//
// Next Step
//
//   Switch over to next step under conditions:
//   or Maximal steptime
//   or Minimal steptime
//           and
//               or no setpoint delta temp
//               or atual value delta temp is ge setpoint deltatemp
//                   and sensor is ok
//           and
// /              or no setpoint max temp above floor
//              or atual value max temp above floor is ge setpoint max temp above floor
//                  and sensor is ok
// 1 Kriterium
      U(    ;
      L     "MAL1S033Par".ActTimeStepProcess.SteptimeActMinOverall; // Steptime in min overall
      L     "MAL1S033Par".StepAct.StepTime_Max; // Target steptime actual step
      >=I   ;
      )     ;
      O(    ;
// 2 Kriterium
      O(    ;
      U(    ;
      L     "MAL1S033Par".StepAct.DeltaTempSwitchpointStep;
      L     0;
//JV230310      >=D
      >D    ; //JV230310
      )     ;
// condition, if analogue input is not damaaged   //
      UN    "G295M".A_3291_BTE07.OutOverflow; //AIR TEMPERATURE ABOVE FLOOR
      UN    "G295M".A_3291_BTE07.OutFaultAI; //AIR TEMPERATURE ABOVE FLOOR
      UN    "G295M".A_3291_BTE01.OutOverflow; //AIR TEMPERATURE BELOW FLOOR
      UN    "G295M".A_3291_BTE01.OutFaultAI; //AIR TEMPERATURE BELOW FLOOR
      U(    ;
      L     "G295M".A_3291_BTE01.OutValueUnits; // act value temperature below floor
      L     "G295M".A_3291_BTE07.OutValueUnits; // act value temperature above floor
      -D    ; // delta temp actual
      L     L#10;
      /D    ;
      L     "MAL1S033Par".StepAct.DeltaTempSwitchpointStep;
      <D    ;
      )     ;
      )     ;
// 3 Kriterium
      O(    ;
      U(    ;
      L     "MAL1S033Par".StepAct.MaxTempAboveFloorStep;
      L     L#0; // 0,0°C is illegally switchpoint for max. temperature
      >D    ;
      )     ;
// condition, if analogue input is not damaaged   // MW R2.1
      UN    "G295M".A_3291_BTE01.OutOverflow; //AIR TEMPERATURE BELOW FLOOR
      UN    "G295M".A_3291_BTE01.OutFaultAI; //AIR TEMPERATURE BELOW FLOOR
      U(    ;
      L     "G295M".A_3291_BTE07.OutValueUnits; // act value temperature above floor
      L     L#10;
      /D    ;
      L     "MAL1S033Par".StepAct.MaxTempAboveFloorStep;
      >=D   ;
      )     ;
      )     ;
// 4 Kriterium
// and min. time
      U(    ;
      L     "MAL1S033Par".ActTimeStepProcess.SteptimeActMinOverall; // Steptime in min overall
//JV210710 Unsinn      L     "MAL1S033Par".RecipeHeader.Cleaning.SPARE_INT0001    // Target steptime actual step
      L     "MAL1S033Par".StepAct.StepTime_Min; // Target steptime actual step //JV210710
      >=I   ;
      )     ;
      )     ;
// and not cooling                                // UK 22.01.07
      UN    "MAL1S033Par".Par.FlagProcess.Cooling_Activ;
// 5 Kriterium
      O(    ;
      U     "MAL1S033Par".Par.FlagProcess.Cooling_Activ;
      U(    ;
      L     "G295M".A_3291_BTE07.OutValueUnits; // act value temperature above floor
      L     L#10;
      /D    ;
      L     "MAL1S033Par".StepAct.TemperaturAboveFloor;
      <=D   ;
      )     ;
      O(    ;
      L     "MAL1S033Par".Par.ParIntMachine.ActualStep;
//JV210710      L     25                          // max. 24 Schritte
      L     27; // max. 26 Schritte   //JV210710
      >=I   ;
      )     ;
      )     ;
// and min. time
      U(    ;
      L     "MAL1S033Par".ActTimeStepProcess.SteptimeActMinOverall; // Steptime in min overall
      L     "MAL1S033Par".StepAct.StepTime_Min; // Target steptime actual step
      >=I   ;
      )     ;
      SPBN  E606;
// send average step data to PIC
      SET   ;
      S     "MAL1S033StepValues".SendData; // send average step data to PIC
// Next step
      L     "MAL1S033Par".Par.ParIntMachine.ActualStep;
      L     "MAL1S033Par".RecipeHeader.NumberOfSteps;
      >I    ;
      SPB   Pedk; // Last step is finished
//BRT20100901 ====> Schritt halten
      U     "MAL1S033Par".Par.FlagProcess.Inf08; // Schritt halten
      SPB   E606;
//BRT20100901 <====
//
      L     "MAL1S033Par".Par.ParIntMachine.ActualStep;
      L     1;
      +I    ;
      T     "MAL1S033Par".Par.ParIntMachine.ActualStep;
      L     0;
      T     "MAL1S033Par".ActTimeStepProcess.SteptimeActMinOverall; // Steptime in min Overall
      SPA   E606;
Pedk: NOP   0; // Process has finished
      SET   ;
      R     "MAL1S033Par".Par.FlagProcess.ProcessActive;
      R     "MAL1S033Par".Par.FlagProcess.Cooling_Activ;
      S     "MAL1S033Par".Par.FlagProcess.ProcessEnd;
//
      L     0; // clear step number
      T     "MAL1S033Par".Par.ParIntMachine.ActualStep;
      T     "MAL1S033Par".StepAct.StepNumber;
E606: NOP   0;
NETWORK
TITLE =ASW_6080: Active step kilning
//
      U     "MAL1S033Par".Par.FlagProcess.ProcessActive;
      SPBN  E608;
// copy stepnr for visu
      L     "MAL1S033Par".Par.ParIntMachine.ActualStep;
      T     "MAL1S033Par".Par.ParIntProcess.ActualStep;
//MW 2010.04.26
      U(    ;
      L     "MAL1S033Par".StepAct.StepTime_Min;
      L     0;
      ==I   ;
      )     ;
      U(    ;
      L     "MAL1S033Par".StepAct.StepTime_Max;
      L     0;
      ==I   ;
      )     ;
      SPB   Nklk;
// basic speed  fans
      L     "MAL1S033Par".StepAct.SpeedVentilatorBasic;
      T     "MAL1S033Par".Par.ParIntProcess.SpeedVentilatorBasic;
// basic position exhaust air flaps
      L     "MAL1S033Par".StepAct.PosExhaustAirFlapBasic; // setpoint from recipe
      L     10; // convert to 0.1%
      *I    ;
      T     "MAL1S033Par".Par.ParIntProcess.PosExhaustAirFlapBasic;
// basic position withering air channel flaps
      L     "MAL1S033Par".StepAct.PosWitheringAirFlapBasic; // setpoint from recipe
      L     10; // convert to 0.1%
      *I    ;
      T     "MAL1S033Par".Par.ParIntProcess.PosWitheringAirFlapBasic;
// basic position recycling air channel flaps
      L     "MAL1S033Par".StepAct.PosRecycleAirFlapBasic; // setpoint from recipe
      L     10; // convert to 0.1%
      *I    ;
      T     "MAL1S033Par".Par.ParIntProcess.PosRecycAirFlapBasic;
      T     "MAL1S033Par".Par.ProcessValue.Value17; // Sollwert Umluftklappen Verbund
//MW 2010.04.26
// basic position fresh air flaps
//      L     "MAL1S033Par".StepAct.PosFreshAirFlapBasic    // setpoint from recipe
      L     0; // 0%
      U     "MAL1S033Par".Par.FlagProcess.ProcessActive;
      UN    "MAL1S033Par".Par.FlagProcess.Cooling_Activ;
      SPB   klk;
      L     100; // 100%
      U     "MAL1S033Par".Par.FlagProcess.ProcessActive;
      U     "MAL1S033Par".Par.FlagProcess.Cooling_Activ;
      SPB   klk;
      SPA   Nklk;
klk:  L     10; // convert to 0.1%
      *I    ;
      T     "MAL1S033Par".Par.ParIntProcess.PosFreshAirFlapBasic;
Nklk: NOP   0;

// Nachlauf der Brenner
//    U     "GCS7_GrCtrlDB".OutEnable[276]    // G276M Heating Kilningbox
      U     "MAL1S033Par".Par.FlagProcess.ProcessActive;
      UN    "MAL1S033Par".Par.FlagProcess.Cooling_Activ;
      =     "MAL1S033Par".Par.FlagProcess.ProgrammSchwelkenDarren;

      U     "MAL1S033Par".Par.FlagProcess.ProgrammSchwelkenDarren;
      L     S5T#1M;
      SA    T     60; // Nachlauf Brenner

      UN    "MAL1S033Par".Par.FlagProcess.ProgrammSchwelkenDarren;
      U     T     60; // Nachlauf Brenner
      =     "MAL1S033Par".Par.FlagProcess1.HilfsRegler_1_Down;
      =     "MAL1S033Par".Par.FlagProcess1.HilfsRegler_2_Down;
      =     "MAL1S033Par".Par.FlagProcess1.HilfsRegler_3_Down;
      =     "MAL1S033Par".Par.FlagProcess1.HilfsRegler_4_Down;

// Sollwert - Istwert vergleich der Temperatur unter der Horde
      L     "MAL1S033Par".StepAct.TemperaturBelowFloor; // setpoint from SCADA
      L     L#10;
      *D    ;
      T     "MAL1S033Par".Par.ProcessValue.TemperaturBelowFloor;

      U     "SYS_Scan0_Tick1min";
      SPBN  NORM;
//- nur alle x Minuten korrigieren ---
      L     "MAL1S033Par".Par.ProcessValue.CorrInterval;
      +     1;
      T     "MAL1S033Par".Par.ProcessValue.CorrInterval;
      L     2; // Korrekturintervall [min]
      >=I   ;
      SPBN  NORM;
      L     0;
      T     "MAL1S033Par".Par.ProcessValue.CorrInterval;

      L     "MAL1S033Par".Par.ProcessValue.TemperaturBelowFloor;
      L     "G295M".A_3291_BTE01.OutValueUnits; // Real-Value Temperature below floor
      -D    ;
      L     50; // Totband in [0.5°C]
      <=D   ;
      SPB   uebe; // wenn größer keine Korrektur
//- zur Sicherheit nicht mehr als 5.0°C zulassen ---
      L     5.000000e+002; // max. Korrektur !
      L     "MAL1S033Par".Par.ProcessValue_Real.SollwertTempKorr;
      <=R   ;
      SPB   uebe;
      L     "MAL1S033Par".Par.ProcessValue_Real.SollwertTempKorr;
      L     1.000000e+000; // Anpassung an Differenz zwischen den PT100
      +R    ;
      T     "MAL1S033Par".Par.ProcessValue_Real.SollwertTempKorr;
uebe: NOP   0;

      L     "MAL1S033Par".Par.ProcessValue.TemperaturBelowFloor;
      L     "G295M".A_3291_BTE01.OutValueUnits; // Real-Value Temperature below floor
      -D    ;
      L     50; // Totband in [0.5°C]
      >=D   ;
      SPB   unte; // wenn kleier keine Korrektur
//- keine negative Korrektur (führt sonst zu Schwingung) ---
      L     0.000000e+000; // keine negative Korrektur !
      L     "MAL1S033Par".Par.ProcessValue_Real.SollwertTempKorr;
      >=R   ;
      SPB   unte;
      L     1.000000e+000; // Anpassung an Differenz zwischen den PT100
      -R    ;
      T     "MAL1S033Par".Par.ProcessValue_Real.SollwertTempKorr;
unte: NOP   0;

//- bei Schrittbegin noch keine Korrektur ---
NORM: L     "MAL1S033Par".ActTimeStepProcess.SteptimeActMinOverall; // Steptime in min overall
      L     8; // Korrekturverzögerung [min]
      >I    ;
      SPB   SET;
      L     0.000000e+000;
      T     "MAL1S033Par".Par.ProcessValue_Real.SollwertTempKorr;
      L     10; // grossen Wert in Intervallzähler vorladen ...
      T     "MAL1S033Par".Par.ProcessValue.CorrInterval; // ... damit nächster 1MinTick gleich wirksam wird

SET:  NOP   0;
      L     "MAL1S033Par".Par.ProcessValue.TemperaturBelowFloor;
      DTR   ;
      L     "MAL1S033Par".Par.ProcessValue_Real.SollwertTempKorr;
      +R    ;
      T     "MAL1S033Par".Par.ProcessValue_Real.T_SOLL_NORM;
      SPA   M641;
      NOP   0;
//- Korrekturfaktor auf "0" setzen ---
      L     0.000000e+000;
      T     "MAL1S033Par".Par.ProcessValue_Real.SollwertTempKorr;
M641: NOP   0;
      SPA   GCPR;

// GCPRO
// setpoint temperature below floor
      NOP   0; // setpoint fans automatic mode
      L     L#0;
      U     "MAL1S033Par".Par.FlagProcess.Cooling_Activ; // switch over to cooling
      SPB   aut1;
      L     "MAL1S033Par".StepAct.TemperaturBelowFloor; // setpoint from SCADA
aut1: NOP   0;
      DTR   ;
      L     1.000000e+001;
      /R    ;
      T     "MAL1S033Par".Par.ProcessValue_Real.T_SOLL_NORM;
// emergency kiln heating
// fan 1
      U(    ;
      L     2#1;
      L     "MAL1S033Par".RecipeHeader.DeselectVentilator; // emergency regime without fan 1
      ==I   ;
      )     ;
      L     "G295M".A_3291_BTE05.OutValuePc; //AIR TEMPERATURE DIFFUSOR FAN 1 :  temperature in diffusor fan 1
      SPBN  c1R1;
      L     "G295M".A_3291_BTE01.OutValuePc; //AIR TEMPERATURE BELOW FLOOR
      L     "G295M".A_3291_BTE05.OutValuePc; //AIR TEMPERATURE DIFFUSOR FAN 1 :  temperature in diffusor fan 2
      <D    ;
      SPBN  c1R1;
      TAK   ;
c1R1: T     "MAL1S033Par".Par.ParIntProcess.ActValueTemperature_R1;
// fan 2
      U(    ;
      L     2#10;
      L     "MAL1S033Par".RecipeHeader.DeselectVentilator; // emergency regime without fan 2
      ==I   ;
      )     ;
      L     "G295M".A_3291_BTE05.OutValuePc; //AIR TEMPERATURE DIFFUSOR FAN 1 :  temperature in diffusor fan 2
      SPBN  c1R2;
      L     "G295M".A_3291_BTE01.OutValuePc; //AIR TEMPERATURE BELOW FLOOR
      L     "G295M".A_3291_BTE05.OutValuePc; //AIR TEMPERATURE DIFFUSOR FAN 1 :  temperature in diffusor fan 1
      <D    ;
      SPBN  c1R2;
      TAK   ;
c1R2: T     "MAL1S033Par".Par.ParIntProcess.ActValueTemperature_R2;

GCPR: NOP   0;
//BRT20100901 ====> Schritt halten, wenn in Rezept aktiviert!!!
      U(    ;
      L     "MAL1S033Par".RecipeHeader.SPARE_DINT004;
      L     L#1; // Schritt halten aktiviert = 1
      ==D   ;
      )     ;
      U(    ;
      L     "G295M".A_3291_BTE07.OutValuePc; // Temperature above floor kiln 2
      L     100;
      /D    ;
      L     "MAL1S033Par".RecipeHeader.SPARE_INT002; // Schaltpunkt für Schritt halten
      >=I   ;
      )     ;
      U(    ;
      U     "MAL1S032".ToASW.InfDataReady; // Kiln 1 bereit
      O     "MAL1S032Par".Par.FlagFunction_1.StepLoading;
      )     ;
      UN    "MAL1S032Par".Par.FlagProcess.ProcessActive;
      UN(   ;
      U     "G271M".A_3125_MXZ01MA.Ma.StStartedFwd;
      U     "G271M".A_3125_TSC01_AF.OutL; // Ventilator 1 dreht mind. 40% SW
      U     "G271M".A_3126_MXZ01MA.Ma.StStartedFwd;
      U     "G271M".A_3126_TSC01_AF.OutL; // Ventilator 2 dreht mind. 40% SW
      )     ;
      S     "MAL1S033Par".Par.FlagProcess.Inf08; // Schritt halten

      U(    ;
      L     "MAL1S033Par".RecipeHeader.SPARE_DINT004;
      L     L#1; // Schritt halten aktiviert = 1
      <>D   ;
      )     ;
      O(    ;
      U     "MAL1S032Par".Par.FlagProcess.ProcessActive;
      U(    ;
      U     "G271M".A_3125_MXZ01MA.Ma.StStartedFwd;
      U     "G271M".A_3125_TSC01_AF.OutL; // Ventilator 1 dreht mind. 40% SW
      O     ;
      U     "G271M".A_3126_MXZ01MA.Ma.StStartedFwd;
      U     "G271M".A_3126_TSC01_AF.OutL; // Ventilator 2 dreht mind. 40% SW
      )     ;
      )     ;
      R     "MAL1S033Par".Par.FlagProcess.Inf08; // Schritt halten
//BRT20100901 <====
// cooling down
      L     "MAL1S033Par".StepAct.CoolingDown;
      L     1;
      ==I   ;
      S     "MAL1S033Par".Par.FlagProcess.Cooling_Activ;
//JV250710 =====>
      L     "MAL1S033Par".Par.ParIntMachine.ActualStep;
      L     24;
      <I    ;
      O(    ; //JV290710 ======>
      L     "MAL1S033Par".StepAct.CoolingDown;
      L     1;
      <>I   ;
      )     ; //JV290710 <=====
      R     "MAL1S033Par".Par.FlagProcess.Cooling_Activ;
//JV250710 <=====
E608: NOP   0;
//BRT20100901 ====> Schritt-Halte-Bit wird nochmals explizit bei Prozess Ende zurückgesetzt!!!
      UN    "MAL1S033Par".Par.FlagProcess.ProcessActive;
      O     "MAL1S033Par".Par.FlagProcess.ProcessEnd;
      R     "MAL1S033Par".Par.FlagProcess.Inf08; // Schritt halten

// Abdarr-Betrieb aktiv
      U(    ;
      L     "MAL1S033Par".Par.ParIntMachine.ActualStep;
      L     "MAL1S032Par".Par.ParIntMachine.ActualStep;
      >I    ;
      )     ;
      UN    "MAL1S033Par".Par.FlagProcess.Cooling_Activ;
      O     "MAL1S032Par".Par.FlagProcess.Cooling_Activ;
//BRT20100830 ====> Bit Abdarr Betrieb Aktiv abhängig von Rezeptwert!
//      =     "MAL1S033Par".Par.FlagProcess.Abdarr_Betrieb_Aktiv
      =     "MAL1S033Par".Par.FlagProcess2.Inf22; // Hilfsbit für Abdarr-Betrieb

      U     "MAL1S033Par".Par.FlagProcess2.Inf22; // Hilfsbit für Abdarr-Betrieb
      U(    ; // Schaltpunkt Schwelken/Darren aus Line Parameter
      L     "G295M".A_3291_BTE07.OutValuePc; // Temperature above floor
      L     L#100;
      /D    ;
//BRT20100901 ====> geändert von Line Parameter nach General in Rezept!!!
//      L     "MAL1Par".Values1.Value04   // Line Parameter
      L     "MAL1S033Par".RecipeHeader.SPARE_INT000; // Rezept Parameter
//BRT20100901 <====
      >=D   ;
      )     ;
      S     "MAL1S033Par".Par.FlagProcess.Abdarr_Betrieb_Aktiv;

      UN    "MAL1S033Par".Par.FlagProcess2.Inf22; // Hilfsbit für Abdarr-Betrieb
      R     "MAL1S033Par".Par.FlagProcess.Abdarr_Betrieb_Aktiv;
//BRT20100830 <====

//BRT20100830 ====> Regelung während Verbundbetrieb!!!
//
      U     "MAL1S033Par".Par.FlagProcess.ProcessActive;
      U     "MAL1S033Par".Par.FlagProcess.Abdarr_Betrieb_Aktiv;
      U(    ;
      L     "MAL1S033Par".Par.ParIntMachine.ActualStep;
      L     "MAL1S033Par".Par.ProcessValue.Value16; // Step-Copy
      >I    ;
      )     ;
      FP    "MAL1S033Par".Par.FlagProcess2.Inf23;
      =     "MAL1S033Par".Par.FlagProcess2.Inf24;

//Einlesen der Rezeptwerte jeden neuen Schritt!
      U     "MAL1S033Par".Par.FlagProcess2.Inf24;
      O(    ;
      L     "MAL1S033Par".RecipeHeader.SPARE_DINT0003;
      L     L#1; // autom. Regelung ON = 1
      <>D   ;
      )     ;
      ON(   ;
      L     "G295M".A_3291_BTE07.OutValuePc; // Temperature above floor kiln 2
      L     5500; // 55°C
      >=I   ;
      )     ;
      SPBN  rd01;
      L     "MAL1S033Par".Par.ParIntMachine.ActualStep;
      T     "MAL1S033Par".Par.ProcessValue.Value16; // Step-Copy

      L     "MAL1S033Par".Par.ParIntProcess.PosRecycAirFlapBasic; // setpoint from recipe
      T     "MAL1S033Par".Par.ProcessValue.Value17; // Sollwert Umluftklappen Verbund

      L     "MAL1S033Par".Par.ParIntProcess.SpeedVentilatorBasic; // setpoint from recipe
      T     "MAL1S033Par".Par.ProcessValue.Value18; // Sollwert Ventilator Verbund
rd01: NOP   0;

//BRT20100903 ====> Verzögerung nach Step-Wechsel bis Regelung aktiv!
      U     "MAL1S033Par".Par.FlagProcess2.Inf24;
      L     S5T#15M;
      SV    T     32;
//BRT20100903 <====

      U     "MAL1S033Par".Par.FlagProcess.ProcessActive;
      U     "MAL1S033Par".Par.FlagProcess.Abdarr_Betrieb_Aktiv;
      U(    ;
      L     "MAL1S033Par".RecipeHeader.SPARE_DINT0003;
      L     L#1; // autom. Regelung ON = 1
      ==D   ;
      )     ;
      UN    T     32; // Verzögerung nach Step-Wechsel   //BRT20100903
      UN    T     33; // alle 5 min kann geregelt werden
      U(    ;
      L     "G295M".A_3291_BTE07.OutValuePc; // Temperature above floor kiln 2
      L     5500; // 55°C
      >=I   ;
      )     ;
      SPBN  nore;
      L     "MAL1S032Par".StepAct.TemperaturBelowFloor;
      L     10;
      -I    ;
      L     10;
      *I    ;
      L     "G269M".A_3191_BTE01.OutValuePc; // Temperature below floor kiln 1
      >I    ;
      SPB   pls1;
      L     "MAL1S032Par".StepAct.TemperaturBelowFloor;
      L     10;
      +I    ;
      L     10;
      *I    ;
      L     "G269M".A_3191_BTE01.OutValuePc; // Temperature below floor kiln 1
      <I    ;
      SPB   mns1;
      SPA   recl;
pls1: NOP   0;
//      L     "MAL1S033Par".Par.ProcessValue.Value17    // Sollwert Umluftklappen Verbund
//      L     50                          // 5%
//      -D
//      T     "MAL1S033Par".Par.ProcessValue.Value17    // Sollwert Umluftklappen Verbund

      L     "MAL1S033Par".Par.ProcessValue.Value18; // Sollwert Ventilator Verbund
      L     L#2; // 2%
      +D    ;
      T     "MAL1S033Par".Par.ProcessValue.Value18; // Sollwert Ventilator Verbund
      SPA   recl;
mns1: NOP   0;
//      L     "MAL1S033Par".Par.ProcessValue.Value17    // Sollwert Umluftklappen Verbund
//      L     50                          // 5%
//      +D
//      T     "MAL1S033Par".Par.ProcessValue.Value17    // Sollwert Umluftklappen Verbund

      L     "MAL1S033Par".Par.ProcessValue.Value18; // Sollwert Ventilator Verbund
      L     L#2; // 2%
      -D    ;
      T     "MAL1S033Par".Par.ProcessValue.Value18; // Sollwert Ventilator Verbund
recl: NOP   0;

//Kontrolle der Regelwerte Umluftklappen Grenzwerte Min/Max
//      L     "MAL1S033Par".Par.ProcessValue.Value17    // Sollwert Umluftklappen Verbund
//      L     "MAL1S033Par".Par.ParIntProcess.PosRecycAirFlapBasic    // setpoint from recipe
//      <D
//      SPB   min1
//      TAK
//min1: T     "MAL1S033Par".Par.ProcessValue.Value17    // Sollwert Umluftklappen Verbund

//      L     "MAL1S033Par".Par.ProcessValue.Value17    // Sollwert Umluftklappen Verbund
//      L     L#900                       // maximum 90%
//      >D
//      SPB   max1
//      TAK
//max1: T     "MAL1S033Par".Par.ProcessValue.Value17    // Sollwert Umluftklappen Verbund

//Kontrolle der Regelwerte Ventilator Grenzwerte Min/max
      L     "MAL1S033Par".Par.ProcessValue.Value18; // Sollwert Ventilator Verbund
      L     L#60; // minimum 60%
      <D    ;
      SPB   min2;
      TAK   ;
min2: T     "MAL1S033Par".Par.ProcessValue.Value18; // Sollwert Ventilator Verbund

      L     "MAL1S033Par".Par.ProcessValue.Value18; // Sollwert Ventilator Verbund
      L     L#100; // maximum 100%
      >D    ;
      SPB   max2;
      TAK   ;
max2: T     "MAL1S033Par".Par.ProcessValue.Value18; // Sollwert Ventilator Verbund
nore: NOP   0;

// 5 min Tick für Regelung
      UN    T     33;
      L     S5T#5M;
      SV    T     33;

//BRT20100830 <====

//BRT20100826 ====> neu mit geregelter Abkühlung!
//
      U     "MAL1S033Par".Par.FlagProcess.Cooling_Activ;
      FP    "MAL1S033Par".Par.FlagProcess2.Inf20;
      =     "MAL1S033Par".Par.FlagProcess2.Inf21;

      U     "MAL1S033Par".Par.FlagProcess2.Inf21;
      O(    ; // in Schritt 25/26 nach Rezeptwert fahren !!!
      L     "MAL1S033Par".Par.ParIntMachine.ActualStep;
      L     24;
      >I    ;
      )     ;
      SPBN  read;
      L     "MAL1S033Par".StepAct.MaxTempAboveFloorStep;
      T     "MAL1S033Par".Par.ProcessValue.Value13; // Schaltpunkt Regelung

      L     "MAL1S033Par".Par.ParIntProcess.PosRecycAirFlapBasic; // setpoint from recipe
      T     "MAL1S033Par".Par.ProcessValue.Value14; // Sollwert Umluftklappen Kühlen

      L     "MAL1S033Par".Par.ParIntProcess.SpeedVentilatorBasic; // setpoint from recipe
      T     "MAL1S033Par".Par.ProcessValue.Value15; // Sollwert Ventilator Kühlen
read: NOP   0;


      L     "G295M".A_3291_BTE07.OutValuePc; // Temperature above floor
      L     L#10;
      /D    ;
      L     "MAL1S033Par".Par.ProcessValue.Value13; // Schaltpunkt Regelung
      <D    ;
      U(    ; // Regelung nur im Schritt 24 !!!
      L     "MAL1S033Par".Par.ParIntMachine.ActualStep;
      L     24;
      ==I   ;
      )     ;
      U     "SYS_Scan0_Tick30s"; //zur Sicherheit
      SPBN  cont;
//neuen Schaltpunkt für nächsten Schritt generieren
      L     "MAL1S033Par".Par.ProcessValue.Value13; // Schaltpunkt Regelung
      L     L#20; // 2,0° C
      -D    ;
      T     "MAL1S033Par".Par.ProcessValue.Value13; // Schaltpunkt Regelung

      L     "MAL1S033Par".Par.ProcessValue.Value14; // Sollwert Umluftklappen Kühlen
      L     L#100; // 10%
      -D    ;
      L     L#0; // Überwachung min. Position
      <=D   ;
      SPB   null;
      TAK   ;
null: T     "MAL1S033Par".Par.ProcessValue.Value14; // Sollwert Umluftklappen Kühlen


      L     "MAL1S033Par".Par.ProcessValue.Value15; // Sollwert Ventilator Kühlen
      L     L#6; // 6%
      +D    ;
      L     L#100; // Überwachung max. Drehzahl
      >=D   ;
      SPB   hdrt;
      TAK   ;
hdrt: T     "MAL1S033Par".Par.ProcessValue.Value15; // Sollwert Ventilator Kühlen

cont: NOP   0;

NETWORK
TITLE =ASW_6090: calculate heat quantity active kilning

      L     L#0;
      U     "MAL1S033Par".Par.FlagProcess.ProcessActive;
      SPBN  n609; // no addition
      SET   ;
      S     "MAL1S033Par".Par.FlagProcess.Inf21; // add heat quantity
      U     "SYS_Scan0_Tick1s"; // scan 1sec
      SPBN  E609;
      L     "MAL1S033Par".Par.ProcessValue_Real.Value05; // heat quantity in kW
      +R    ;
      T     "MAL1S033Par".Par.ProcessValue_Real.Value05;
      SPA   E609;
n609: NOP   0;
      U     "MAL1S033Par".Par.FlagProcess.Inf21; // add heat quantity
      SPBN  E609;
      R     "MAL1S033Par".Par.FlagProcess.Inf21; // add heat quantity
      L     "MAL1S033Par".Par.ProcessValue_Real.Value05;
      L     3.600000e+003;
      /R    ; // from kWs to kWh
      L     1.000000e+003;
      /R    ; // from kWh to MWh
      RND   ;
      T     "MAL1S033Par".Par.ProcessValue_Real.Value06; // result to batch potokoll
      L     0.000000e+000; // clear calculator
      T     "MAL1S033Par".Par.ProcessValue_Real.Value05;
E609: NOP   0;
NETWORK
TITLE =ASW_7000: Step loading kilning
//
      U     "MAL1S033".ToASW.InfDataReady;
      U     "MAL1S033".PCRead.Step.StWait;
      U     "MAL1S033".PCWrite.ExtFuncOn.StartLoading; // PIC command "start loading"
      S     "MAL1S033Par".Par.FlagFunction_1.StepLoading; // Step loading
      R     "MAL1S033Par".Par.FlagMachine.ImpulsNullstellung;
      R     "MAL1S033Par".Par.FlagMachine.CmdTurnRevAfterLoading;
      R     "MAL1S033Par".Par.FlagMachine.CmdTurnFwdAfterLoading;
//MW 2010.04.26
      R     "MAL1S033Par".Par.FlagFunction_0.MerkerBeladenGestartetFP;
//
      SET   ;
      R     "MAL1S033".PCWrite.ExtFuncOn.StartLoading; // PIC command "start loading"
//
//MW 2010.04.26
      U     "MAL1S033Par".Par.FlagFunction_1.StepLoading;
      U     "MAL1S033".ToASW.InfSameBatchPrevSec;
      S     "MAL1S033Par".Par.FlagFunction_0.MerkerBeladenGestartetFP;
//
      U     "MAL1S033".ToASW.InfDataReady;
      U     "MAL1S033".PCRead.Step.StActive;
      U     "MAL1S033Par".Par.FlagFunction_1.StepLoading; // Step loading
      SPB   e71;
      R     "MAL1S033Par".Par.Switches1.StaOn00; // LiftingPositionRound_1
      R     "MAL1S033Par".Par.Switches1.StaOn01; // LiftingPositionRound_2
      R     "MAL1S033Par".Par.Switches1.StaOn02; // LiftingPositionRound_3
      R     "MAL1S033Par".Par.Switches1.StaOn03; // LiftingPositionRound_4
      R     "MAL1S033Par".Par.Switches1.StaOn04; // LiftingPositionRound_5
      R     "MAL1S033Par".Par.Switches1.StaOn05; // LiftingPositionRound_6
e71:  NOP   0;
      U     "MAL1S033".ToASW.InfDataReady;
      U     "MAL1S033".PCRead.Step.StActive;
      U     "MAL1S033Par".Par.FlagFunction_1.StepLoading; // Step loading
//MW 2010.04.26      UN    "MAL1S033Par".Par.FlagFunction_1.FinishLoading
//MW 2010.04.26      UN    "MAL1S033Par".Par.FlagFunction_1.LoadEnd
      SPBN  E700;
      U(    ;
      U(    ;
      L     "G292M".A_3211_MXZ41MA.Ma.OutPositionAngle;
      L     3460; // 346.0°
      >=I   ;
      )     ;
      O     ;
      U(    ;
      L     "G292M".A_3211_MXZ41MA.Ma.OutCntRound;
      L     L#1;
      >=D   ;
      )     ;
      )     ;
      U     "MAL1S033Par".Par.FlagFunction_1.StepLoading;
      =     "MAL1S033Par".Par.FlagFunction_0.ReducedSpeed;
//
      L     "MAL1S033Par".RecipeHeader.Loading.LiftingPositionRound_3;
      L     20; // 20°
      -I    ;
      T     "MAL1S033Par".Par.ParIntMachine.LiftingPositionRound_4;
      L     "MAL1S033Par".RecipeHeader.Loading.LoadingLevelRound_3;
      L     "MAL1S033Par".RecipeHeader.Loading.OffsetLevelNextRound;
      +I    ;
      T     "MAL1S033Par".Par.ParIntMachine.LoadingLevelRound_4;
//
      L     "MAL1S033Par".Par.ParIntMachine.LiftingPositionRound_4;
      L     20; // 20°
      -I    ;
      T     "MAL1S033Par".Par.ParIntMachine.LiftingPositionRound_5;
      L     "MAL1S033Par".Par.ParIntMachine.LoadingLevelRound_4;
      L     "MAL1S033Par".RecipeHeader.Loading.OffsetLevelNextRound;
      +I    ;
      T     "MAL1S033Par".Par.ParIntMachine.LoadingLevelRound_5;
//
      L     "MAL1S033Par".Par.ParIntMachine.LiftingPositionRound_5;
      L     20; // 20°
      -I    ;
      T     "MAL1S033Par".Par.ParIntMachine.LiftingPositionRound_6;
      L     "MAL1S033Par".Par.ParIntMachine.LoadingLevelRound_5;
      L     "MAL1S033Par".RecipeHeader.Loading.OffsetLevelNextRound;
      +I    ;
      T     "MAL1S033Par".Par.ParIntMachine.LoadingLevelRound_6;
//
      L     3600;
      L     "G292M".A_3211_MXZ41MA.Ma.Par.ParTolPosition;
      -I    ;
      L     "G292M".A_3211_MXZ41MA.Ma.OutPositionAngle;
      <=I   ;
      SPB   E700;
//MW 2010.04.26
      L     3600;
      L     "G292M".A_3211_MXZ41MA.Ma.Par.ParTolPosition;
      -I    ;
      L     "G292M".A_3211_MXZ41MA.Ma.OutPositionAngle;
      <=I   ;
      U     "G292M".A_3211_MXZ41MA.A_3211_MXZ41.OutpRunFwd;
      SPB   E700;
//
//MW 2010.04.26      L     "G292M".A_3211_MXZ41MA.Ma.OutPositionAngle
//MW 2010.04.26      L     0
//MW 2010.04.26      <I
//MW 2010.04.26//      <=I
//MW 2010.04.26
      L     "G292M".A_3211_MXZ41MA.Ma.OutPositionAngle;
      L     0;
      <=I   ;
      U     "G292M".A_3211_MXZ41MA.A_3211_MXZ41.OutpRunFwd;
      SPB   E700;
//
      L     "G292M".A_3211_MXZ41MA.Ma.OutPositionAngle;
      L     10;
      /I    ;
      T     "MAL1S033Par".Par.MachineValue.ISTWERT_FAHRANTRIEB_POSI;
//
      U     "MAL1S033Par".Par.FlagFunction_1.StepLoading; // Step loading
      FP    "MAL1S033Par".Par.Switches1.StaOn08;
      =     "MAL1S033Par".Par.Switches1.StaOn09; // scan start loading
      U     "MAL1S033Par".Par.Switches1.StaOn09; // scan start loading
      SPBN  e72;
      R     "MAL1S033Par".Par.Switches1.StaOn00; // LiftingPositionRound_1
      R     "MAL1S033Par".Par.Switches1.StaOn01; // LiftingPositionRound_2
      R     "MAL1S033Par".Par.Switches1.StaOn02; // LiftingPositionRound_3
      R     "MAL1S033Par".Par.Switches1.StaOn03; // LiftingPositionRound_4
      R     "MAL1S033Par".Par.Switches1.StaOn04; // LiftingPositionRound_5
      R     "MAL1S033Par".Par.Switches1.StaOn05; // LiftingPositionRound_6
//
e72:  NOP   0;
//
      U(    ;
      L     "G292M".A_3211_MXZ41MA.Ma.OutCntRound;
      L     L#0;
      ==D   ;
      )     ;
      U(    ;
      L     "MAL1S033Par".Par.MachineValue.ISTWERT_FAHRANTRIEB_POSI;
      L     "MAL1S033Par".RecipeHeader.Loading.LiftingPositionRound_1;
      <I    ;
      )     ;
      S     "MAL1S033Par".Par.Switches1.StaOn00; // LiftingPositionRound_1
//
      U(    ;
      L     "G292M".A_3211_MXZ41MA.Ma.OutCntRound;
      L     L#0;
      ==D   ;
      )     ;
      U(    ;
      L     "MAL1S033Par".Par.MachineValue.ISTWERT_FAHRANTRIEB_POSI;
      L     "MAL1S033Par".RecipeHeader.Loading.LiftingPositionRound_1;
      >=I   ;
      )     ;
      U(    ;
      L     "MAL1S033Par".Par.MachineValue.ISTWERT_FAHRANTRIEB_POSI;
      L     3550; // 355.0° --> Ruckeln am Nullpunkt abfangen
      <=I   ;
      )     ;
      S     "MAL1S033Par".Par.Switches1.StaOn01; // LiftingPositionRound_2
//
      U     "MAL1S033Par".Par.Switches1.StaOn01; // LiftingPositionRound_2
      R     "MAL1S033Par".Par.Switches1.StaOn00; // LiftingPositionRound_1
//
      U(    ;
      L     "G292M".A_3211_MXZ41MA.Ma.OutCntRound;
      L     L#1;
      ==D   ;
      )     ;
      U(    ;
      L     "MAL1S033Par".Par.MachineValue.ISTWERT_FAHRANTRIEB_POSI;
      L     "MAL1S033Par".RecipeHeader.Loading.LiftingPositionRound_2;
      >=I   ;
      )     ;
//MW 2010.04.26
      U(    ;
      L     "MAL1S033Par".Par.MachineValue.ISTWERT_FAHRANTRIEB_POSI;
      L     "MAL1S033Par".RecipeHeader.Loading.LiftingPositionRound_1;
      <I    ;
      )     ;
      S     "MAL1S033Par".Par.Switches1.StaOn02; // LiftingPositionRound_3
//
      U     "MAL1S033Par".Par.Switches1.StaOn02; // LiftingPositionRound_3
      R     "MAL1S033Par".Par.Switches1.StaOn01; // LiftingPositionRound_2
      R     "MAL1S033Par".Par.Switches1.StaOn00; // LiftingPositionRound_1
//
      U(    ;
      L     "G292M".A_3211_MXZ41MA.Ma.OutCntRound;
      L     L#2;
      ==D   ;
      )     ;
      U(    ;
      L     "MAL1S033Par".Par.MachineValue.ISTWERT_FAHRANTRIEB_POSI;
      L     "MAL1S033Par".RecipeHeader.Loading.LiftingPositionRound_3;
      >=I   ;
      )     ;
//MW 2010.04.26
      U(    ;
      L     "MAL1S033Par".Par.MachineValue.ISTWERT_FAHRANTRIEB_POSI;
      L     "MAL1S033Par".RecipeHeader.Loading.LiftingPositionRound_2;
      <I    ;
      )     ;
      S     "MAL1S033Par".Par.Switches1.StaOn03; // LiftingPositionRound_4
//
      U     "MAL1S033Par".Par.Switches1.StaOn03; // LiftingPositionRound_4
      R     "MAL1S033Par".Par.Switches1.StaOn02; // LiftingPositionRound_3
      R     "MAL1S033Par".Par.Switches1.StaOn01; // LiftingPositionRound_2
      R     "MAL1S033Par".Par.Switches1.StaOn00; // LiftingPositionRound_1
      U(    ;
      L     "G292M".A_3211_MXZ41MA.Ma.OutCntRound;
      L     L#3;
      ==D   ;
      )     ;
      U(    ;
      L     "MAL1S033Par".Par.MachineValue.ISTWERT_FAHRANTRIEB_POSI;
      L     "MAL1S033Par".Par.ParIntMachine.LiftingPositionRound_4;
      >=I   ;
      )     ;
//MW 2010.04.26
      U(    ;
      L     "MAL1S033Par".Par.MachineValue.ISTWERT_FAHRANTRIEB_POSI;
      L     "MAL1S033Par".RecipeHeader.Loading.LiftingPositionRound_3;
      <I    ;
      )     ;
      S     "MAL1S033Par".Par.Switches1.StaOn04; // LiftingPositionRound_5
//
      U     "MAL1S033Par".Par.Switches1.StaOn04; // LiftingPositionRound_5
      R     "MAL1S033Par".Par.Switches1.StaOn03; // LiftingPositionRound_4
      R     "MAL1S033Par".Par.Switches1.StaOn02; // LiftingPositionRound_3
      R     "MAL1S033Par".Par.Switches1.StaOn01; // LiftingPositionRound_2
      R     "MAL1S033Par".Par.Switches1.StaOn00; // LiftingPositionRound_1
      U(    ;
      L     "G292M".A_3211_MXZ41MA.Ma.OutCntRound;
      L     L#4;
      ==D   ;
      )     ;
      U(    ;
      L     "MAL1S033Par".Par.MachineValue.ISTWERT_FAHRANTRIEB_POSI;
      L     "MAL1S033Par".Par.ParIntMachine.LiftingPositionRound_5;
      >=I   ;
      )     ;
//MW 2010.04.26
      U(    ;
      L     "MAL1S033Par".Par.MachineValue.ISTWERT_FAHRANTRIEB_POSI;
      L     "MAL1S033Par".RecipeHeader.Loading.LiftingPositionRound_4;
      <I    ;
      )     ;
      S     "MAL1S033Par".Par.Switches1.StaOn05; // LiftingPositionRound_6
//
      U     "MAL1S033Par".Par.Switches1.StaOn05; // LiftingPositionRound_6
      R     "MAL1S033Par".Par.Switches1.StaOn04; // LiftingPositionRound_5
      R     "MAL1S033Par".Par.Switches1.StaOn03; // LiftingPositionRound_4
      R     "MAL1S033Par".Par.Switches1.StaOn02; // LiftingPositionRound_3
      R     "MAL1S033Par".Par.Switches1.StaOn01; // LiftingPositionRound_2
      R     "MAL1S033Par".Par.Switches1.StaOn00; // LiftingPositionRound_1
      U     "MAL1S033Par".Par.Switches1.StaOn00; // LiftingPositionRound_1
      SPB   Rnd1;
      U     "MAL1S033Par".Par.Switches1.StaOn01; // LiftingPositionRound_2
      SPB   Rnd2;
      U     "MAL1S033Par".Par.Switches1.StaOn02; // LiftingPositionRound_3
      SPB   Rnd3;
      U     "MAL1S033Par".Par.Switches1.StaOn03; // LiftingPositionRound_4
      SPB   Rnd4;
      U     "MAL1S033Par".Par.Switches1.StaOn04; // LiftingPositionRound_5
      SPB   Rnd5;
      U     "MAL1S033Par".Par.Switches1.StaOn05; // LiftingPositionRound_6
      SPB   Rnd6;
      SPA   E700;
Rnd1: NOP   0;
      L     "MAL1S033Par".RecipeHeader.Loading.LoadingLevelRound_1;
      L     "G291M".A_3211_MXZ21_31MA.Ma.Par.ParTolPosition;
      +I    ;
      T     "MAL1S033Par".Par.MachineValue.SOLLWERT_HUBZUG1_HOEHE;
      T     "MAL1S033Par".Par.MachineValue.SOLLWERT_HUBZUG2_HOEHE;
      L     "MAL1S033Par".RecipeHeader.Loading.LoadingSpeed_1;
      T     "MAL1S033Par".Par.MachineValue.SollwertFahrantrieb;
      SPA   E700;
Rnd2: NOP   0;
      L     "MAL1S033Par".RecipeHeader.Loading.LoadingLevelRound_2;
      L     "G291M".A_3211_MXZ21_31MA.Ma.Par.ParTolPosition;
      +I    ;
      T     "MAL1S033Par".Par.MachineValue.SOLLWERT_HUBZUG1_HOEHE;
      T     "MAL1S033Par".Par.MachineValue.SOLLWERT_HUBZUG2_HOEHE;
      L     "MAL1S033Par".RecipeHeader.Loading.LoadingSpeed_2;
      T     "MAL1S033Par".Par.MachineValue.SollwertFahrantrieb;
      SPA   E700;
Rnd3: NOP   0;
      L     "MAL1S033Par".RecipeHeader.Loading.LoadingLevelRound_3;
      L     "G291M".A_3211_MXZ21_31MA.Ma.Par.ParTolPosition;
      +I    ;
      T     "MAL1S033Par".Par.MachineValue.SOLLWERT_HUBZUG1_HOEHE;
      T     "MAL1S033Par".Par.MachineValue.SOLLWERT_HUBZUG2_HOEHE;
      L     "MAL1S033Par".RecipeHeader.Loading.LoadingSpeed_3;
      T     "MAL1S033Par".Par.MachineValue.SollwertFahrantrieb;
      SPA   E700;
Rnd4: NOP   0;
      L     "MAL1S033Par".Par.ParIntMachine.LoadingLevelRound_4;
      L     "G291M".A_3211_MXZ21_31MA.Ma.Par.ParTolPosition;
      +I    ;
      T     "MAL1S033Par".Par.MachineValue.SOLLWERT_HUBZUG1_HOEHE;
      T     "MAL1S033Par".Par.MachineValue.SOLLWERT_HUBZUG2_HOEHE;
//      L     "MAL1S033Par".RecipeHeader.Loading.LoadingSpeed_3
      L     87; // 87%
      T     "MAL1S033Par".Par.MachineValue.SollwertFahrantrieb;
      SPA   E700;
Rnd5: NOP   0;
      L     "MAL1S033Par".Par.ParIntMachine.LoadingLevelRound_5;
      L     "G291M".A_3211_MXZ21_31MA.Ma.Par.ParTolPosition;
      +I    ;
      T     "MAL1S033Par".Par.MachineValue.SOLLWERT_HUBZUG1_HOEHE;
      T     "MAL1S033Par".Par.MachineValue.SOLLWERT_HUBZUG2_HOEHE;
//      L     "MAL1S033Par".RecipeHeader.Loading.LoadingSpeed_3
      L     87; // 87%
      T     "MAL1S033Par".Par.MachineValue.SollwertFahrantrieb;
      SPA   E700;
Rnd6: NOP   0;
      L     "MAL1S033Par".Par.ParIntMachine.LoadingLevelRound_6;
      L     "G291M".A_3211_MXZ21_31MA.Ma.Par.ParTolPosition;
      +I    ;
      T     "MAL1S033Par".Par.MachineValue.SOLLWERT_HUBZUG1_HOEHE;
      T     "MAL1S033Par".Par.MachineValue.SOLLWERT_HUBZUG2_HOEHE;
//      L     "MAL1S033Par".RecipeHeader.Loading.LoadingSpeed_3
      L     87; // 87%
      T     "MAL1S033Par".Par.MachineValue.SollwertFahrantrieb;
      SPA   E700;
E700: NOP   0;
NETWORK
TITLE =Sub 7010: Kilning  loading finished
//      L     0;
//      L     "MAL1S033".ToSSW.InPrevSecDB;
//      ==I   ;
//      SPB   fin;
//      O(;
//      U     "MAL1S017Par".Par.FlagFunction_1.FinishUnloading;
//      U     "MAL1S033".PCWrite.ExtFuncOn.FinishLoading; // PIC command "finish
//loading"
//      O       "MAL1S017Par".Par.FlagFunction_1.StepCleaning;
//      U     "MAL1S017".PCRead.Step.StEmptied;
//      U(    ;
//      AUF   "MAL1S017";
//      L DBNO;
//      L     "MAL1S033".ToSSW.InPrevSecDB;
//      ==I;
//      )     ;
//      )     ;
//      O(;
//      U     "MAL1S018Par".Par.FlagFunction_1.FinishUnloading;
//      U     "MAL1S033".PCWrite.ExtFuncOn.FinishLoading; // PIC command "finish
//loading"
//      O       "MAL1S018Par".Par.FlagFunction_1.StepCleaning;
//      U     "MAL1S018".PCRead.Step.StEmptied;
//      U(    ;
//      AUF   "MAL1S018";
//      L DBNO;
//      L     "MAL1S033".ToSSW.InPrevSecDB;
//      ==I;
//      )     ;
//      )     ;
//      O(;
//      U     "MAL1S019Par".Par.FlagFunction_1.FinishUnloading;
//      U     "MAL1S033".PCWrite.ExtFuncOn.FinishLoading; // PIC command "finish
//loading"
//      O       "MAL1S019Par".Par.FlagFunction_1.StepCleaning;
//      U     "MAL1S019".PCRead.Step.StEmptied;
//      U(    ;
//      AUF   "MAL1S019";
//      L DBNO;
//      L     "MAL1S033".ToSSW.InPrevSecDB;
//      ==I;
//      )     ;
//      )     ;
//      O(;
//      U     "MAL1S020Par".Par.FlagFunction_1.FinishUnloading;
//      U     "MAL1S033".PCWrite.ExtFuncOn.FinishLoading; // PIC command "finish
//loading"
//      O       "MAL1S020Par".Par.FlagFunction_1.StepCleaning;
//      U     "MAL1S020".PCRead.Step.StEmptied;
//      U(    ;
//      AUF   "MAL1S020";
//      L DBNO;
//      L     "MAL1S033".ToSSW.InPrevSecDB;
//      ==I;
//      )     ;
//      )     ;
//      O(;
//      U     "MAL1S021Par".Par.FlagFunction_1.FinishUnloading;
//      U     "MAL1S033".PCWrite.ExtFuncOn.FinishLoading; // PIC command "finish
//loading"
//      O       "MAL1S021Par".Par.FlagFunction_1.StepCleaning;
//      U     "MAL1S021".PCRead.Step.StEmptied;
//      U(    ;
//      AUF   "MAL1S021";
//      L DBNO;
//      L     "MAL1S033".ToSSW.InPrevSecDB;
//      ==I;
//      )     ;
//      )     ;
//      O(;
//      U     "MAL1S022Par".Par.FlagFunction_1.FinishUnloading;
//      U     "MAL1S033".PCWrite.ExtFuncOn.FinishLoading; // PIC command "finish
//loading"
//      O       "MAL1S022Par".Par.FlagFunction_1.StepCleaning;
//      U     "MAL1S022".PCRead.Step.StEmptied;
//      U(    ;
//      AUF   "MAL1S022";
//      L DBNO;
//      L     "MAL1S033".ToSSW.InPrevSecDB;
//      ==I;
//      )     ;
//      )     ;
//      O(;
//      U     "MAL1S023Par".Par.FlagFunction_1.FinishUnloading;
//      U     "MAL1S033".PCWrite.ExtFuncOn.FinishLoading; // PIC command "finish l
//oading"
//      O       "MAL1S023Par".Par.FlagFunction_1.StepCleaning;
//      U     "MAL1S023".PCRead.Step.StEmptied;
//      U(    ;
//      AUF   "MAL1S023";
//      L DBNO;
//      L     "MAL1S033".ToSSW.InPrevSecDB;
//      ==I;
//      )     ;
//      )     ;
//      O(;
//      U     "MAL1S024Par".Par.FlagFunction_1.FinishUnloading;
//      U     "MAL1S033".PCWrite.ExtFuncOn.FinishLoading; // PIC command "finish
//loading"
//      O       "MAL1S024Par".Par.FlagFunction_1.StepCleaning;
//      U     "MAL1S024".PCRead.Step.StEmptied;
//      U(    ;
//      AUF   "MAL1S024";
//      L DBNO;
//      L     "MAL1S033".ToSSW.InPrevSecDB;
//      ==I;
//      )     ;
//      )     ;
//      O(    ;
//      U     "MAL1S033Par".Par.FlagFunction_1.StepLoading; // Step loading
//      UN    "MAL1S033".ToASW.InfSameJobPrevSec;
//      U     "MAL1S033".PCWrite.ExtFuncOn.FinishLoading; // PIC command "finish l
//oading"
//      )     ;
//      U     "MAL1S033".ToASW.InfDataReady;
//      U     "MAL1S033".PCRead.Step.StActive;
//      S     "MAL1S033Par".Par.FlagFunction_1.LoadEnd;
////
//      U     "MAL1S033".PCWrite.ExtFuncOn.FinishLoading; // PIC command "finish
//loading"
//      R     "MAL1S033".PCWrite.ExtFuncOn.FinishLoading; // PIC command "finish l
//oading"
////
//      U     "MAL1S033Par".Par.FlagFunction_1.LoadEnd;
//      U     "MAL1S033Par".Par.FlagFunction_1.StepLoading; // Step loading
//      FP    "MAL1S033Par".Par.FlagFunction_0.ImpulsSollposition;
//      =     "MAL1S033Par".Par.FlagFunction_0.MerkerSollpositionFP;
//      U     "MAL1S033Par".Par.FlagFunction_0.MerkerSollpositionFP;
//      SPBN  fin;
//      L     WinCoS_BIW01_09PLC1BIW01_02.Ma.OutPositionAngle;
//      L     "MAL1S033Par".Par.ParIntProcess.LoadingOverlap;
//      +I    ;
//      T     WinCoS_BIW01_09PLC1BIW01_02.Ma.InPositionTarget;
////???      SET
////???      S     "PLC1BIW01_02".TurningTo_Parkposition    //
//WinCoS_BIW01_09PLC1BIW01_02..Ma.InAdjusting
//// Beladehöhe speichern
//      L     "MAL1S033Par".Par.MachineValue.SOLLWERT_HUBZUG1_HOEHE;
//      T     "MAL1S033Par".Par.ParIntMachine.LastLoadingLevel; // saved loading
//value
//fin:  NOP   0;
//E701: NOP   0;
// Grundschicht vollständig bedeckt
//MW 2010.04.26
      U(    ;
      L     "G292M".A_3211_MXZ41MA.Ma.OutPositionAngle;
      L     3580; // 358.0°
      <I    ;
      )     ;
      U(    ;
// Die Position bei IBN ermitteln!
      L     "G292M".A_3211_MXZ41MA.Ma.OutPositionAngle;
//MW 2010.04.26      L     3564                        // 356.4°
      L     3540; // 354.0°
      >=I   ;
      )     ;
      U     "MAL1S033Par".Par.FlagFunction_1.StepLoading;
      U     "G292M".A_3211_MXZ41MA.Ma.InEnableFwd;
      S     "MAL1S033Par".Par.FlagFunction_1.LoadFirstPartEnd;
      S     "MAL1S033Par".Par.FlagProcess.Product_Inside;

      U     "MAL1S033Par".Par.FlagProcess.ProcessActive;
      U     "MAL1S033Par".Par.FlagFunction_1.FinishLoading;
      O     "MAL1S033Par".Par.FlagFunction_1.StepUnloading;
      O     "MAL1S033".PCRead.Step.StIdling; // "SecDB".PCRead.Step.StIdling
      R     "MAL1S033Par".Par.FlagFunction_1.LoadFirstPartEnd;

      L     0;
      L     "MAL1S033".ToSSW.InPrevSecDB;
      ==I   ;
//MW 2010.04.26      SPB   fin
//MW 2010.04.26
      SPB   suki;
      O(    ;
      U     "MAL1S017Par".Par.FlagFunction_1.FinishUnloading;
      O     "MAL1S017Par".Par.FlagFunction_1.StepCleaning; // Step cleaning
      O     "MAL1S017Par".Par.FlagFunction_1.FinishCleaning;
      U     "MAL1S017".PCRead.Step.StEmptied;
      ON    "MAL1S017".ToASW.InfDataReady; //JV070810
      U     "MAL1S033".PCWrite.ExtFuncOn.FinishLoading; // PIC command "finish loading"
      U(    ;
      AUF   "MAL1S017";
      L     DBNO;
      L     "MAL1S033".ToSSW.InPrevSecDB;
      ==I   ;
      )     ;
      )     ;
      O(    ;
      U     "MAL1S018Par".Par.FlagFunction_1.FinishUnloading;
      O     "MAL1S018Par".Par.FlagFunction_1.StepCleaning; // Step cleaning
      O     "MAL1S018Par".Par.FlagFunction_1.FinishCleaning;
      U     "MAL1S018".PCRead.Step.StEmptied;
      ON    "MAL1S018".ToASW.InfDataReady; //JV070810
      U     "MAL1S033".PCWrite.ExtFuncOn.FinishLoading; // PIC command "finish loading"
      U(    ;
      AUF   "MAL1S018";
      L     DBNO;
      L     "MAL1S033".ToSSW.InPrevSecDB;
      ==I   ;
      )     ;
      )     ;
      O(    ;
      U     "MAL1S019Par".Par.FlagFunction_1.FinishUnloading;
      O     "MAL1S019Par".Par.FlagFunction_1.StepCleaning; // Step cleaning
      O     "MAL1S019Par".Par.FlagFunction_1.FinishCleaning;
      U     "MAL1S019".PCRead.Step.StEmptied;
      ON    "MAL1S019".ToASW.InfDataReady; //JV070810
      U     "MAL1S033".PCWrite.ExtFuncOn.FinishLoading; // PIC command "finish loading"
      U(    ;
      AUF   "MAL1S019";
      L     DBNO;
      L     "MAL1S033".ToSSW.InPrevSecDB;
      ==I   ;
      )     ;
      )     ;
      O(    ;
      U     "MAL1S020Par".Par.FlagFunction_1.FinishUnloading;
      O     "MAL1S020Par".Par.FlagFunction_1.StepCleaning; // Step cleaning
      O     "MAL1S020Par".Par.FlagFunction_1.FinishCleaning;
      U     "MAL1S020".PCRead.Step.StEmptied;
      ON    "MAL1S020".ToASW.InfDataReady; //JV070810
      U     "MAL1S033".PCWrite.ExtFuncOn.FinishLoading; // PIC command "finish loading"
      U(    ;
      AUF   "MAL1S020";
      L     DBNO;
      L     "MAL1S033".ToSSW.InPrevSecDB;
      ==I   ;
      )     ;
      )     ;
      O(    ;
      U     "MAL1S021Par".Par.FlagFunction_1.FinishUnloading;
      O     "MAL1S021Par".Par.FlagFunction_1.StepCleaning; // Step cleaning
      O     "MAL1S021Par".Par.FlagFunction_1.FinishCleaning;
      U     "MAL1S021".PCRead.Step.StEmptied;
      ON    "MAL1S021".ToASW.InfDataReady; //JV070810
      U     "MAL1S033".PCWrite.ExtFuncOn.FinishLoading; // PIC command "finish loading"
      U(    ;
      AUF   "MAL1S021";
      L     DBNO;
      L     "MAL1S033".ToSSW.InPrevSecDB;
      ==I   ;
      )     ;
      )     ;
      O(    ;
      U     "MAL1S022Par".Par.FlagFunction_1.FinishUnloading;
      O     "MAL1S022Par".Par.FlagFunction_1.StepCleaning; // Step cleaning
      O     "MAL1S022Par".Par.FlagFunction_1.FinishCleaning;
      U     "MAL1S022".PCRead.Step.StEmptied;
      ON    "MAL1S022".ToASW.InfDataReady; //JV070810
      U     "MAL1S033".PCWrite.ExtFuncOn.FinishLoading; // PIC command "finish loading"
      U(    ;
      AUF   "MAL1S022";
      L     DBNO;
      L     "MAL1S033".ToSSW.InPrevSecDB;
      ==I   ;
      )     ;
      )     ;
      O(    ;
      U     "MAL1S023Par".Par.FlagFunction_1.FinishUnloading;
      O     "MAL1S023Par".Par.FlagFunction_1.StepCleaning; // Step cleaning
      O     "MAL1S023Par".Par.FlagFunction_1.FinishCleaning;
      U     "MAL1S023".PCRead.Step.StEmptied;
      ON    "MAL1S023".ToASW.InfDataReady; //JV070810
      U     "MAL1S033".PCWrite.ExtFuncOn.FinishLoading; // PIC command "finish loading"
      U(    ;
      AUF   "MAL1S023";
      L     DBNO;
      L     "MAL1S032".ToSSW.InPrevSecDB;
      ==I   ;
      )     ;
      )     ;
      O(    ;
      U     "MAL1S024Par".Par.FlagFunction_1.FinishUnloading;
      O     "MAL1S024Par".Par.FlagFunction_1.StepCleaning; // Step cleaning
      O     "MAL1S024Par".Par.FlagFunction_1.FinishCleaning;
      U     "MAL1S024".PCRead.Step.StEmptied;
      ON    "MAL1S024".ToASW.InfDataReady; //JV070810
      U     "MAL1S033".PCWrite.ExtFuncOn.FinishLoading; // PIC command "finish loading"
      U(    ;
      AUF   "MAL1S024";
      L     DBNO;
      L     "MAL1S033".ToSSW.InPrevSecDB;
      ==I   ;
      )     ;
      )     ;
suki: NOP   0;
      O(    ;
      U     "MAL1S033Par".Par.FlagFunction_1.StepLoading; // Step loading
      UN    "MAL1S033".ToASW.InfSameJobPrevSec;
      U     "MAL1S033".PCWrite.ExtFuncOn.FinishLoading; // PIC command "finish loading"
      )     ;
      U     "MAL1S033".ToASW.InfDataReady;
      U     "MAL1S033".PCRead.Step.StActive;
      U     "MAL1S033Par".Par.FlagFunction_1.LoadFirstPartEnd;
      S     "MAL1S033Par".Par.FlagFunction_1.LoadEnd;
      R     "MAL1S017".PCWrite.ExtFuncOn.FinishCleanSurface; // PIC command "finish unloading"
      R     "MAL1S018".PCWrite.ExtFuncOn.FinishCleanSurface; // PIC command "finish unloading"
      R     "MAL1S019".PCWrite.ExtFuncOn.FinishCleanSurface; // PIC command "finish unloading"
      R     "MAL1S020".PCWrite.ExtFuncOn.FinishCleanSurface; // PIC command "finish unloading"
      R     "MAL1S021".PCWrite.ExtFuncOn.FinishCleanSurface; // PIC command "finish unloading"
      R     "MAL1S022".PCWrite.ExtFuncOn.FinishCleanSurface; // PIC command "finish unloading"
      R     "MAL1S023".PCWrite.ExtFuncOn.FinishCleanSurface; // PIC command "finish unloading"
      R     "MAL1S024".PCWrite.ExtFuncOn.FinishCleanSurface; // PIC command "finish unloading"

//
//MW 2010.04.26      U     "MAL1S033".PCWrite.ExtFuncOn.FinishLoading    // PIC command "finish loading"
//MW 2010.04.26      R     "MAL1S033".PCWrite.ExtFuncOn.FinishLoading    // PIC command "finish loading"
//
      U     "MAL1S033Par".Par.FlagFunction_1.LoadEnd;
      U     "MAL1S033Par".Par.FlagFunction_1.StepLoading; // Step loading
      FP    "MAL1S033Par".Par.FlagFunction_0.ImpulsSollposition;
      =     "MAL1S033Par".Par.FlagFunction_0.MerkerSollpositionFP;
      U     "MAL1S033Par".Par.FlagFunction_0.MerkerSollpositionFP;
      SPBN  fin;
      L     "G292M".A_3211_MXZ41MA.Ma.OutPositionAngle;
      L     "MAL1S033Par".Par.ParIntProcess.LoadingOverlap;
//MW 2010.04.26
      +I    ;
      L     3600; // 360,0°
      >=I   ;
      SPBN  SOZ1;
      -I    ;
      SPA   SOZ2;
SOZ1: NOP   0;
      TAK   ;
SOZ2: NOP   0;
      T     "G292M".A_3211_MXZ41MA.Ma.InPositionTarget;
      SET   ;
//MW 2010.04.26      S     "G292M".TurningTo_Parkposition
      S     "MAL1S033Par".Par.FlagMachine.WEGMESSUNG_0_FLAG;

// Extra Planierrunde wenn der Fahrantrieb ueber 346° beim Beladen Ende war
      L     "G292M".A_3211_MXZ41MA.Ma.OutPositionAngle;
      L     3460; // 346,0 °
      >I    ;
      S     "G292M".Turning_One_Round_More;

// Beladehöhe speichern
      L     "MAL1S033Par".Par.MachineValue.SOLLWERT_HUBZUG1_HOEHE;
      T     "MAL1S033Par".Par.ParIntMachine.LastLoadingLevel; // saved loading value
fin:  NOP   0;

// Hubzüge erst auf der Parkposition abheben
//MW 2010.04.26      U     "G292M".TurningTo_Parkposition
//MW 2010.04.26      FN    "G291M".USW8
//MW 2010.04.26      =     "G291M".USW9

//MW 2010.04.26      U     "G291M".USW9
//MW 2010.04.26      O
//MW 2010.04.26      U     "MAL1S033Par".Par.FlagFunction_1.FinishLoading
//MW 2010.04.26      U(
//MW 2010.04.26     U     "G292M".A_3211_MXZ41MA.A_3211_BZS43.StCtoTrue    // sensor zero point
//MW 2010.04.26      O     "G292M".A_3211_MXZ41MA.A_3211_BZS43.StTrue    // sensor zero point
//MW 2010.04.26      )
//MW 2010.04.26      SPBN  auf
//MW 2010.04.26      L     "G291M".A_3211_MXZ21_31MA.Ma.Par.ParPositionTopLeftUnits    //LIFTING DRIVE
//MW 2010.04.26      L     150
//MW 2010.04.26      +I
//MW 2010.04.26      T     "MAL1S033Par".Par.MachineValue.SOLLWERT_HUBZUG1_HOEHE
//MW 2010.04.26      L     "G291M".A_3211_MXZ21_31MA.Ma.Par.ParPositionTopRightUnits    //LIFTING DRIVE
//MW 2010.04.26      L     150
//MW 2010.04.26      +I
//MW 2010.04.26      T     "MAL1S033Par".Par.MachineValue.SOLLWERT_HUBZUG2_HOEHE
//MW 2010.04.26      L     1
//MW 2010.04.26      T     "G291M".A_3211_MXZ21_31MA.Ma.Par.ParTolPosition
//MW 2010.04.26 auf:  NOP   0
      NOP   0;
NETWORK
TITLE =ASW_6080: Processtime Kilning
//      CALL  "SSA_MH_ProcessTime_Fct" , DB1017
//       InfDataReady :="MAL1S017".ToASW.InfDataReady
//       ProzessActive:="MAL1S017Par".Par.FlagProcess.ProcessActive
//       InStartTime  :="MAL1S017Par".Prozesstime.Starttime
//       OutStartTime :="MAL1S017Par".Prozesstime.Starttime
//       ProcessTime  :="MAL1S017Par".Prozesstime
//
      CALL "SSA_MH_ProcessTime_Fct" , DB  1033 (
           InfDataReady             := "MAL1S033".ToASW.InfDataReady,
           ProzessActive            := "MAL1S033Par".Par.FlagProcess.ProcessActive,
           InStartTime              := "MAL1S033Par".Processtime.StartTime,
           OutStartTime             := "MAL1S033Par".Processtime.StartTime,
           ProcessTime              := "MAL1S033Par".Processtime);

NETWORK
TITLE =Sub 7020: Step start process kilning
//      U     "MAL1S033".ToASW.InfDataReady
//      U     "MAL1S033".PCRead.Step.StActive
////      U       "MAL1S033".PCWrite.ExtFuncOn.StartProcess    // PIC command
//"start process kilning"
//      U     "MAL1S033Par".Par.FlagFunction_1.LoadEnd
//
//      U     "G292M".A_3211_MXZ41MA.A_3211_BZS43.StTrue    // sensor zero point
//      U     "G291M".A_3211_MXZ21_31MA.A_3211_BZS23.InpTrue
//      U     "G291M".A_3211_MXZ21_31MA.A_3211_BZS33.InpTrue
//
//      O(
//      UN    "MAL1S033".SecNom.Par1On.Cmd01    // With Loading
//      UN    "MAL1S033".ToASW.InfSameBatchPrevSec
//      U     "MAL1S033".ToASW.InfDataReady
//      U     "MAL1S033".PCRead.Step.StActive
//      )
//
//      S     "MAL1S033Par".Par.FlagFunction_1.FinishLoading    // start process
//kilning
//      R     "MAL1S033Par".Par.FlagFunction_1.LoadEnd
////
//      U     "MAL1S033".PCWrite.ExtFuncOn.StartProcess    // PIC command "start
//process kilning"
//      R     "MAL1S033".PCWrite.ExtFuncOn.StartProcess    // PIC command "start
//process kilning"
////
//      U     "G292M".A_3211_MXZ41MA.Ma.StAdjusted
//      O     "G292M".A_3211_MXZ41MA.Ma.OutAdjusted
//      U     "MAL1S033Par".Par.FlagFunction_1.FinishLoading    // start process
//kilning
//      O     "MAL1S033Par".Par.FlagProcess.ProcessActive
//      SPBN  E702
//      L     "G291M".A_3211_MXZ21_31MA.Ma.Par.ParPositionTopLeftUnits
////LIFTING DRIVE
//      L     50                          //jk
//      +I
//      T     "MAL1S033Par".Par.MachineValue.SOLLWERT_HUBZUG1_HOEHE
//      L     "G291M".A_3211_MXZ21_31MA.Ma.Par.ParPositionTopRightUnits
////LIFTING DRIVE
//      L     50                          //jk
//      +I
//      T     "MAL1S033Par".Par.MachineValue.SOLLWERT_HUBZUG2_HOEHE
//      L     1
//      T     "G291M".A_3211_MXZ21_31MA.Ma.Par.ParTolPosition
//
//E702: NOP   0
//
//      U     "G292M".TurningTo_Parkposition
//      SPBN  E703
//      U(
//      L     "G292M".A_3211_MXZ41MA.Ma.OutPositionAngle
//      L     3500
//      >=I
//      )
//      SPBN  E703
//      L     10                          // 10% speed to parkposition
//      T     "MAL1S033Par".Par.MachineValue.SollwertFahrantrieb
//E703: NOP   0
//
//      U     "G292M".TurningTo_Parkposition
//      SPBN  E704
//      U(
//      L     "G292M".A_3211_MXZ41MA.Ma.OutPositionAngle
//      L     3500
//      <I
//      )
//      SPBN  E704
//      L     87                          // 87% speed to parkposition
//      T     "MAL1S033Par".Par.MachineValue.SollwertFahrantrieb
//E704: NOP   0
//
//MW 2010.04.26
      U     "MAL1S033".ToASW.InfDataReady;
      U     "MAL1S033".PCRead.Step.StActive;
      U     "MAL1S033Par".Par.FlagFunction_1.LoadEnd;
      U     "G292M".A_3211_MXZ41MA.Ma.StAdjusted; // travelling drive on target position
//-Without loading---
      O(    ;
      UN    "MAL1S033".SecNom.Par1On.Cmd01; // With Loading
      UN    "MAL1S033".ToASW.InfSameBatchPrevSec;
      U     "MAL1S033".ToASW.InfDataReady;
      U     "MAL1S033".PCRead.Step.StActive;
      )     ;
      O(    ;
      U     "MAL1S033".PCWrite.ExtFuncOn.FinishLoading; // PIC command "finish loading"
      U     "MAL1S033Par".Par.FlagFunction_1.LoadEnd;
      UN    "MAL1S033".ToASW.InfSameBatchPrevSec;
      U     "MAL1S033".ToASW.InfDataReady;
      U     "MAL1S033".PCRead.Step.StActive;
      )     ;
      S     "MAL1S033Par".Par.FlagFunction_1.FinishLoading; // start process kilning
      R     "MAL1S033Par".Par.FlagFunction_1.LoadEnd;
//MW 2010.04.23
      S     "MAL1S033".PCRead.Status.StaLoaded;
//
      U     "MAL1S033".PCWrite.ExtFuncOn.FinishLoading; // PIC command "finish loading"
      R     "MAL1S033".PCWrite.ExtFuncOn.FinishLoading; // PIC command "finish loading"
//
//-With loading---
      U(    ;
      U     "G292M".A_3211_MXZ41MA.Ma.StAdjusted;
      O     "G292M".A_3211_MXZ41MA.Ma.OutAdjusted;
      U     "MAL1S033Par".Par.FlagFunction_1.FinishLoading; // start process kilning
      )     ;
//-Without loading---
      O(    ;
      UN    "MAL1S033".SecNom.Par1On.Cmd01; // With Loading
      UN    "MAL1S033".ToASW.InfSameBatchPrevSec;
      U     "MAL1S033".PCRead.Step.StReady;
      U     "MAL1S033Par".Par.FlagProcess.ProcessActive;
      )     ;
      O(    ;
      U     "MAL1S033".PCRead.Step.StReady;
      U     "MAL1S033Par".Par.FlagProcess.ProcessActive;
      UN    "MAL1S033Par".Par.FlagFunction_1.StepLoading;
      UN    "MAL1S033Par".Par.FlagFunction_1.FinishLoading;
      UN    "MAL1S033Par".Par.FlagFunction_1.LoadEnd;
      UN    "MAL1S033Par".Par.FlagMachine.WEGMESSUNG_0_FLAG;
      )     ;
      SPB   pPos;
      SPA   E702;
pPos: NOP   0;
      L     "G291M".A_3211_MXZ21_31MA.Ma.Par.ParPositionTopLeftUnits; //LIFTING DRIVE
      L     50;
      +I    ;
      T     "MAL1S033Par".Par.MachineValue.SOLLWERT_HUBZUG1_HOEHE;
      L     "G291M".A_3211_MXZ21_31MA.Ma.Par.ParPositionTopRightUnits; //LIFTING DRIVE
      L     50;
      +I    ;
      T     "MAL1S033Par".Par.MachineValue.SOLLWERT_HUBZUG2_HOEHE;
      L     3;
      T     "G291M".A_3211_MXZ21_31MA.Ma.Par.ParTolPosition;
E702: NOP   0;

NETWORK
TITLE =ASW_8000:  Step unloading kilning
//      UN    "MAL1S033Par".Par.FlagFunction_1.StepUnloading    // Step Unloading
//      R     "MAL1S033Par".Par.FlagFunction_0.OverlapSaved    // Ueberlappung
//erfasst
////
//      U     "MAL1S033".ToASW.InfDataReady
//      U     "MAL1S033".PCRead.Step.StEmptying
//      U(
//      L     "MAL1S033Par".RecipeHeader.Unloading.StartUnloadAuto
////StartUnloadAuto = 0
//      L     1
//      <>I
//      U     "MAL1S033".PCWrite.ExtFuncOn.StartUnLoading    // PIC command
//"start
//unloading"
//      O
//      U(
//      L     "MAL1S033Par".RecipeHeader.Unloading.StartUnloadAuto
////StartUnloadAuto = 10
//      L     1
//      ==I
//      )
//      UN    "G297M".A_3225_TSC01_AF.OutL    // 30% Ventilatordrehzahl
//      UN    "G297M".A_3226_TSC01_AF.OutL    // 30% Ventilatordrehzahl
//      )
//      S     "MAL1S033Par".Par.FlagFunction_1.StepUnloading    // Step Unloading
//      R     "MAL1S033Par".Par.FlagMachine.ImpulsNullstellung
//      R     "MAL1S023Par".Par.FlagMachine.WEGMESSUNG_0
//      R     DB923.DBX  148.0            // FP
//      R     "MAL1S033Par".Par.FlagMachine.CmdTurnRevAfterUnloading
//      R     "MAL1S033Par".Par.FlagMachine.CmdTurnFwdAfterUnloading
////
//      SET
//      R     "MAL1S033".PCWrite.ExtFuncOn.StartUnLoading    // PIC command
//"start
//unloading"
////
//      U     "MAL1S033".ToASW.InfDataReady
//      U     "MAL1S033".PCRead.Step.StEmptying
//      U     "MAL1S033Par".Par.FlagFunction_1.StepUnloading    // Step Unloading
//      SPBN  e800
//      L     "MAL1S033Par".Par.ParIntMachine.LastLoadingLevel    // saved
//loading
//value
//      T     "MAL1S033Par".Par.ParIntMachine.FUELLHOEHE_PRODUKT
////
//      U(
//      L     "G291M".A_3211_MXZ21_31MA.Ma.OutPositionLeft
//      L     "MAL1S033Par".Par.ParIntMachine.FUELLHOEHE_PRODUKT
//      >I
//      )
//      O(
//      L     "G291M".A_3211_MXZ21_31MA.Ma.OutPositionRight
//      L     "MAL1S033Par".Par.ParIntMachine.FUELLHOEHE_PRODUKT
//      >I
//      )
//      UN(
//      U(
//      L     "G291M".A_3211_MXZ21_31MA.Ma.OutPositionLeft
//      L     "MAL1S033Par".Par.MachineValue.SOLLWERT_HUBZUG1_HOEHE
//      <=I
//      )
//      U(
//      L     "G291M".A_3211_MXZ21_31MA.Ma.OutPositionRight
//      L     "MAL1S033Par".Par.MachineValue.SOLLWERT_HUBZUG1_HOEHE
//      <=I
//      )
//      )
//      =     "MAL1S033Par".Par.FlagFunction_0.ScrewAboveProductLayer    //
//HubzuegeUeberProdukt
////
////- Letzte Entladehoehe erreicht ---
//      U(
//      L     "MAL1S033Par".Par.MachineValue.SOLLWERT_HUBZUG1_HOEHE
//      L     0
//      <=I
//      )
//      U(
//      L     "MAL1S033Par".Par.MachineValue.SOLLWERT_HUBZUG1_HOEHE
//      L     "G291M".A_3211_MXZ21_31MA.Ma.InPositionTarget
//      ==I
//      )
//      U     "G291M".A_3211_MXZ21_31MA.Ma.StAdjusted
//      U     "MAL1S033Par".Par.FlagFunction_1.StepUnloading    // Step Unloading
//      FP    "MAL1S033Par".Par.FlagFunction_0.UnloadLevelReachedFP    //
//UnloadLevelReachedFP
//      =     "MAL1S033Par".Par.FlagFunction_0.ImpulsUnloadLevelReached    //
//ImpulsUnloadLevelReached
//      UN    "MAL1S033Par".Par.FlagFunction_0.ImpulsUnloadLevelReached    //
//ImpulsUnloadLevelReached
//      O     "MAL1S033Par".Par.FlagFunction_0.OverlapSaved    // Ueberlappung
//erfasst
//      SPB   over
//      L     "G292M".A_3211_MXZ41MA.Ma.OutCntRound
//      L     1
//      +I
//      T     "MAL1S033Par".Par.ParIntProcess.UnloadungRounds
////
//      L     "G292M".A_3211_MXZ41MA.Ma.OutPositionAngle
//      L     3600                        // 360,0°
//      >=I
//      SPBN  soz1
//      -I
//      SPA   soz2
//soz1: NOP   0
//      TAK
//soz2: NOP   0
//      L     100                         // 10,0°
//      +I
//      T     "MAL1S033Par".Par.ParIntProcess.UnloadingOverlap
//      T     "G292M".A_3211_MXZ41MA.Ma.InPositionTarget
//      S     "MAL1S033Par".Par.FlagFunction_0.OverlapSaved    // Ueberlappung
//erfasst
//over: NOP   0
//      U(
//      L     "G292M".A_3211_MXZ41MA.Ma.OutCntRound
//      L     L#0
//      ==D
//      )
//      SPB   rnd1
//      L     "G292M".A_3211_MXZ41MA.Ma.OutCntRound
//      L     L#1
//      ==D
//      SPB   rnd2
//      L     "G292M".A_3211_MXZ41MA.Ma.OutCntRound
//      L     L#2
//      >=D
//      SPB   rnd3
//      SPA   e801
//rnd1: NOP   0
//      L     "MAL1S033Par".RecipeHeader.Loading.LiftingPositionRound_3
//      T     "MAL1S033Par".Par.MachineValue.SOLLWERT_HUBZUG1_HOEHE
//      T     "MAL1S033Par".Par.MachineValue.SOLLWERT_HUBZUG2_HOEHE
//      L     1
//      T     "G291M".A_3211_MXZ21_31MA.Ma.Par.ParTolPosition
//      L     "MAL1S033Par".RecipeHeader.Unloading.UnLoadingSpeed_1
//      T     "MAL1S033Par".Par.MachineValue.SollwertFahrantrieb
//      SPA   e801
//rnd2: NOP   0
//      L     "MAL1S033Par".RecipeHeader.Loading.LiftingPositionRound_4
//      T     "MAL1S033Par".Par.MachineValue.SOLLWERT_HUBZUG1_HOEHE
//      T     "MAL1S033Par".Par.MachineValue.SOLLWERT_HUBZUG2_HOEHE
//      L     1
//      T     "G291M".A_3211_MXZ21_31MA.Ma.Par.ParTolPosition
//      L     "MAL1S033Par".RecipeHeader.Unloading.UnLoadingSpeed_2
//      T     "MAL1S033Par".Par.MachineValue.SollwertFahrantrieb
//      SPA   e801
//rnd3: NOP   0
//      L     "MAL1S033Par".RecipeHeader.Loading.LiftingPositionRound_5
//      T     "MAL1S033Par".Par.MachineValue.SOLLWERT_HUBZUG1_HOEHE
//      T     "MAL1S033Par".Par.MachineValue.SOLLWERT_HUBZUG2_HOEHE
//      L     1
//      T     "G291M".A_3211_MXZ21_31MA.Ma.Par.ParTolPosition
//      L     "MAL1S033Par".RecipeHeader.Unloading.UnLoadingSpeed_3
//      T     "MAL1S033Par".Par.MachineValue.SollwertFahrantrieb
//      SPA   e801
//
//e801: NOP   0
//      U     "MAL1S033".ToASW.InfDataReady
//      U     "MAL1S033".PCRead.Step.StEmptying
//      U     "MAL1S033Par".Par.FlagFunction_1.StepUnloading    // Step Unloading
//      U(
//      L     "G292M".A_3211_MXZ41MA.Ma.OutCntRound
//      L     "MAL1S033Par".Par.ParIntProcess.UnloadungRounds
//      >=I
//      )
//      U     "G291M".A_3211_MXZ21_31MA.Ma.StAdjusted
//      U     "G292M".A_3211_MXZ41MA.Ma.StAdjusted
//      S     "MAL1S033Par".Par.FlagFunction_1.FinishUnloading
//
//      U     "MAL1S033".ToASW.InfDataReady
//      U     "MAL1S033".PCRead.Step.StEmptying
//      U     "MAL1S033Par".Par.FlagFunction_1.FinishUnloading
//      SPBN  e800
//      L     "G291M".A_3211_MXZ21_31MA.Ma.Par.ParPositionTopLeftUnits
//      L     50
//      +I
//      T     "MAL1S033Par".Par.MachineValue.SOLLWERT_HUBZUG1_HOEHE
//      L     "G291M".A_3211_MXZ21_31MA.Ma.Par.ParPositionTopRightUnits
//      L     50
//      +I
//      T     "MAL1S033Par".Par.MachineValue.SOLLWERT_HUBZUG2_HOEHE
//      L     1
//      T     "G291M".A_3211_MXZ21_31MA.Ma.Par.ParTolPosition
//
//      L     0
//      T     "MAL1S033Par".Par.ParIntMachine.LastLoadingLevel    // saved
//loading
//value
//      T     "MAL1S033Par".Par.ParIntMachine.FUELLHOEHE_PRODUKT
//e800: NOP   0
////
//// --> Wie bei der Bank Avangard
//      U     "MAL1S033Par".Par.FlagFunction_1.StepUnloading
//      U     "MAL1S033Par".Par.FlagFunction_1.FinishUnloading
//      FP    DB923.DBX  148.0
//      =     DB923.DBX  148.1
//      SPBN  TAU1
//      L     "G292M".A_3211_MXZ41MA.Ma.OutPositionAngle
//      L     1800
//      <I
//      S     "MAL1S033Par".Par.FlagMachine.CmdTurnRevAfterUnloading
//      L     "G292M".A_3211_MXZ41MA.Ma.OutPositionAngle
//      L     1800
//      >=I
//      S     "MAL1S033Par".Par.FlagMachine.CmdTurnFwdAfterUnloading
//TAU1: NOP   0
//      U     "MAL1S033Par".Par.FlagMachine.CmdTurnRevAfterUnloading
//      O     "MAL1S033Par".Par.FlagMachine.CmdTurnFwdAfterUnloading
//      U     "MAL1S033Par".Par.FlagFunction_1.FinishUnloading
//      U     "G293M".A_3211_MXZ11.StStopped
//      U     "G291M".A_3211_MXZ21_31MA.Ma.OutHigherMinPos
//      U(
//      U     "G291M".A_3211_MXZ21_31MA.A_3211_BZS33.InpTrue
//      U     "G291M".A_3211_MXZ21_31MA.A_3211_BZS23.InpTrue
//      O     "G291M".A_3211_MXZ21_31MA.Ma.StAdjusted
//      )
//      S     "MAL1S033Par".Par.FlagMachine.WEGMESSUNG_0
////
//      U     "MAL1S033".ToASW.InfDataReady
//      U     "MAL1S033Par".Par.FlagFunction_1.FinishUnloading
//      U     "MAL1S033Par".Par.FlagMachine.WEGMESSUNG_0
//      SPBN  TAU2
////    L       "MAL1S033Par".RecipeHeader.Cleaning.CleaningSpeed_1
//      L     30                          // 30%
//      T     "MAL1S033Par".Par.MachineValue.SollwertFahrantrieb
//TAU2: NOP   0
//      NOP   0
//
//MW 2010.04.26
      UN    "MAL1S033Par".Par.FlagFunction_1.StepUnloading; // Step Unloading
      R     "MAL1S033Par".Par.FlagFunction_0.OverlapSaved; // Ueberlappung erfasst
//
      U     "MAL1S033".ToASW.InfDataReady;
      U     "MAL1S033".PCRead.Step.StEmptying;
      U(    ;
      L     "MAL1S033Par".RecipeHeader.Unloading.StartUnloadAuto; //StartUnloadAuto = 0
      L     1;
      <>I   ;
      U     "MAL1S033".PCWrite.ExtFuncOn.StartUnLoading; // PIC command "start unloading"
      O     ;
      U(    ;
      L     "MAL1S033Par".RecipeHeader.Unloading.StartUnloadAuto; //StartUnloadAuto = 10
      L     1;
      ==I   ;
      )     ;
      UN    "G297M".A_3225_TSC01_AF.OutL; // 30% Ventilatordrehzahl
      UN    "G297M".A_3226_TSC01_AF.OutL; // 30% Ventilatordrehzahl
      )     ;
      S     "MAL1S033Par".Par.FlagFunction_1.StepUnloading; // Step Unloading
      R     "MAL1S033Par".Par.FlagMachine.ImpulsNullstellung;
      R     "MAL1S023Par".Par.FlagMachine.WEGMESSUNG_0;
      R     DB923.DBX  148.0; // FP
      R     "MAL1S033Par".Par.FlagMachine.CmdTurnRevAfterUnloading;
      R     "MAL1S033Par".Par.FlagMachine.CmdTurnFwdAfterUnloading;
//
      SET   ;
      R     "MAL1S033".PCWrite.ExtFuncOn.StartUnLoading; // PIC command "start unloading"
//
      U     "MAL1S033".ToASW.InfDataReady;
      U     "MAL1S033".PCRead.Step.StEmptying;
      U     "MAL1S033Par".Par.FlagFunction_1.StepUnloading; // Step Unloading
      SPBN  e800;
//-Start process without loading---
      L     "MAL1S033Par".Par.ParIntMachine.LastLoadingLevel; // saved loading value
      L     0;
      ==I   ;
      L     "MAL1S033Par".RecipeHeader.Loading.LoadingLevelRound_3;
      SPB   LLL;
//-Start process with loading---
      L     "MAL1S033Par".Par.ParIntMachine.LastLoadingLevel; // saved loading value
LLL:  T     "MAL1S033Par".Par.ParIntMachine.FUELLHOEHE_PRODUKT;
//
      U(    ;
      L     "G291M".A_3211_MXZ21_31MA.Ma.OutPositionLeft;
      L     "MAL1S033Par".Par.ParIntMachine.FUELLHOEHE_PRODUKT;
      >I    ;
      )     ;
      O(    ;
      L     "G291M".A_3211_MXZ21_31MA.Ma.OutPositionRight;
      L     "MAL1S033Par".Par.ParIntMachine.FUELLHOEHE_PRODUKT;
      >I    ;
      )     ;
      UN(   ;
      U(    ;
      L     "G291M".A_3211_MXZ21_31MA.Ma.OutPositionLeft;
      L     "MAL1S033Par".Par.MachineValue.SOLLWERT_HUBZUG1_HOEHE;
      <=I   ;
      )     ;
      U(    ;
      L     "G291M".A_3211_MXZ21_31MA.Ma.OutPositionRight;
      L     "MAL1S033Par".Par.MachineValue.SOLLWERT_HUBZUG1_HOEHE;
      <=I   ;
      )     ;
      )     ;
      =     "MAL1S033Par".Par.FlagFunction_0.ScrewAboveProductLayer; // HubzuegeUeberProdukt
//
//- Letzte Entladehoehe erreicht ---
      U(    ;
      L     "MAL1S033Par".Par.MachineValue.SOLLWERT_HUBZUG1_HOEHE;
      L     0;
      <=I   ;
      )     ;
      U(    ;
      L     "MAL1S033Par".Par.MachineValue.SOLLWERT_HUBZUG1_HOEHE;
      L     "G291M".A_3211_MXZ21_31MA.Ma.InPositionTarget;
      ==I   ;
      )     ;
      U     "G291M".A_3211_MXZ21_31MA.Ma.StAdjusted;
      U     "MAL1S033Par".Par.FlagFunction_1.StepUnloading; // Step Unloading
      FP    "MAL1S033Par".Par.FlagFunction_0.UnloadLevelReachedFP; // UnloadLevelReachedFP
      =     "MAL1S033Par".Par.FlagFunction_0.ImpulsUnloadLevelReached; // ImpulsUnloadLevelReached
      UN    "MAL1S033Par".Par.FlagFunction_0.ImpulsUnloadLevelReached; // ImpulsUnloadLevelReached
      O     "MAL1S033Par".Par.FlagFunction_0.OverlapSaved; // Ueberlappung erfasst
      SPB   over;
      L     "G292M".A_3211_MXZ41MA.Ma.OutCntRound;
      L     1;
      +I    ;
      T     "MAL1S033Par".Par.ParIntProcess.UnloadungRounds;
//
      L     "G292M".A_3211_MXZ41MA.Ma.OutPositionAngle;
      L     3600; // 360,0°
      >=I   ;
      SPBN  soz1;
      -I    ;
      SPA   soz2;
soz1: NOP   0;
      TAK   ;
soz2: NOP   0;
//BRT20101018 ====> Overlapping nur noch 5°!!!
//      L     100                         // 10,0°
      L     50; // 5,0°
//<==== BRT20101018
      +I    ;
      T     "MAL1S033Par".Par.ParIntProcess.UnloadingOverlap;
      T     "G292M".A_3211_MXZ41MA.Ma.InPositionTarget;
      S     "MAL1S033Par".Par.FlagFunction_0.OverlapSaved; // Ueberlappung erfasst
over: NOP   0;
      L     "MAL1S033Par".RecipeHeader.Unloading.UnLoadingSpeed_2; //JV290710
      T     "MAL1S033Par".RecipeHeader.Unloading.UnLoadingSpeed_3; //JV290710
//-Only ONE unloading round---  //MW 2010.04.26
// 2 unloading rounds JV290710
//      SPA   rnd1
      U(    ;
      L     "G292M".A_3211_MXZ41MA.Ma.OutCntRound;
      L     L#0;
      ==D   ;
      )     ;
      SPB   rnd1;
      L     "G292M".A_3211_MXZ41MA.Ma.OutCntRound;
      L     L#1;
      ==D   ;
      SPB   rnd2;
      L     "G292M".A_3211_MXZ41MA.Ma.OutCntRound;
      L     L#2;
      >=D   ;
      SPB   rnd3;
      SPA   e801;
rnd1: NOP   0;
      L     "MAL1S033Par".RecipeHeader.Unloading.UnLoadingLevelRound_1;
      T     "MAL1S033Par".Par.MachineValue.SOLLWERT_HUBZUG1_HOEHE;
      T     "MAL1S033Par".Par.MachineValue.SOLLWERT_HUBZUG2_HOEHE;
      L     1;
      T     "G291M".A_3211_MXZ21_31MA.Ma.Par.ParTolPosition;
      L     "MAL1S033Par".RecipeHeader.Unloading.UnLoadingSpeed_1;
      T     "MAL1S033Par".Par.MachineValue.SollwertFahrantrieb;
      SPA   e801;
rnd2: NOP   0;
//JV280710      L     "MAL1S033Par".RecipeHeader.Unloading.UnLoadingLevelRound_2
      L     0; //JV280710   last unloading round
      T     "MAL1S033Par".Par.MachineValue.SOLLWERT_HUBZUG1_HOEHE;
      T     "MAL1S033Par".Par.MachineValue.SOLLWERT_HUBZUG2_HOEHE;
//JV280710      L     1
      L     0; //JV280710
      T     "G291M".A_3211_MXZ21_31MA.Ma.Par.ParTolPosition;
      L     "MAL1S033Par".RecipeHeader.Unloading.UnLoadingSpeed_2;
      T     "MAL1S033Par".Par.MachineValue.SollwertFahrantrieb;
      SPA   e801;
rnd3: NOP   0;
      L     "MAL1S033Par".RecipeHeader.Unloading.UnLoadingLevelRound_3;
      T     "MAL1S033Par".Par.MachineValue.SOLLWERT_HUBZUG1_HOEHE;
      T     "MAL1S033Par".Par.MachineValue.SOLLWERT_HUBZUG2_HOEHE;
      L     1;
      T     "G291M".A_3211_MXZ21_31MA.Ma.Par.ParTolPosition;
      L     "MAL1S033Par".RecipeHeader.Unloading.UnLoadingSpeed_3;
      T     "MAL1S033Par".Par.MachineValue.SollwertFahrantrieb;
      SPA   e801;

e801: NOP   0;
      U     "MAL1S033".ToASW.InfDataReady;
      U     "MAL1S033".PCRead.Step.StEmptying;
      U     "MAL1S033Par".Par.FlagFunction_1.StepUnloading; // Step Unloading
      U(    ;
      L     "G292M".A_3211_MXZ41MA.Ma.OutCntRound;
      L     "MAL1S033Par".Par.ParIntProcess.UnloadungRounds;
      >=I   ;
      )     ;
      U     "G291M".A_3211_MXZ21_31MA.Ma.StAdjusted;
      U     "G292M".A_3211_MXZ41MA.Ma.StAdjusted;
      S     "MAL1S033Par".Par.FlagFunction_1.FinishUnloading;
//MW 2010.04.26
      R     "MAL1S033Par".Par.FlagProcess.Product_Inside;

      U     "MAL1S033".ToASW.InfDataReady;
      U     "MAL1S033".PCRead.Step.StEmptying;
      U     "MAL1S033Par".Par.FlagFunction_1.FinishUnloading;
      SPBN  e800;
      L     "G291M".A_3211_MXZ21_31MA.Ma.Par.ParPositionTopLeftUnits;
      L     50;
      +I    ;
      T     "MAL1S033Par".Par.MachineValue.SOLLWERT_HUBZUG1_HOEHE;
      L     "G291M".A_3211_MXZ21_31MA.Ma.Par.ParPositionTopRightUnits;
      L     50;
      +I    ;
      T     "MAL1S033Par".Par.MachineValue.SOLLWERT_HUBZUG2_HOEHE;
      L     1;
      T     "G291M".A_3211_MXZ21_31MA.Ma.Par.ParTolPosition;

//MW 2010.04.26      L     0
//MW 2010.04.26      T     "MAL1S033Par".Par.ParIntMachine.LastLoadingLevel    // saved loading value
//MW 2010.04.26      T     "MAL1S033Par".Par.ParIntMachine.FUELLHOEHE_PRODUKT
e800: NOP   0;
//
// --> Wie bei der Bank Avangard
      U     "MAL1S033Par".Par.FlagFunction_1.StepUnloading;
      U     "MAL1S033Par".Par.FlagFunction_1.FinishUnloading;
      FP    DB923.DBX  148.0;
      =     DB923.DBX  148.1;
      SPBN  TAU1;
      L     "G292M".A_3211_MXZ41MA.Ma.OutPositionAngle;
      L     1800;
      <I    ;
      S     "MAL1S033Par".Par.FlagMachine.CmdTurnRevAfterUnloading;
      L     "G292M".A_3211_MXZ41MA.Ma.OutPositionAngle;
      L     1800;
      >=I   ;
      S     "MAL1S033Par".Par.FlagMachine.CmdTurnFwdAfterUnloading;
TAU1: NOP   0;
      U     "MAL1S033Par".Par.FlagMachine.CmdTurnRevAfterUnloading;
      O     "MAL1S033Par".Par.FlagMachine.CmdTurnFwdAfterUnloading;
      U     "MAL1S033Par".Par.FlagFunction_1.FinishUnloading;
      U     "G293M".A_3211_MXZ11.StStopped;
      U     "G291M".A_3211_MXZ21_31MA.Ma.OutHigherMinPos;
      U(    ;
      U     "G291M".A_3211_MXZ21_31MA.A_3211_BZS33.InpTrue;
      U     "G291M".A_3211_MXZ21_31MA.A_3211_BZS23.InpTrue;
      O     "G291M".A_3211_MXZ21_31MA.Ma.StAdjusted;
      )     ;
      S     "MAL1S033Par".Par.FlagMachine.WEGMESSUNG_0;
//
      U     "MAL1S033".ToASW.InfDataReady;
      U     "MAL1S033Par".Par.FlagFunction_1.FinishUnloading;
      U     "MAL1S033Par".Par.FlagMachine.WEGMESSUNG_0;
      SPBN  TAU2;
//    L     "MAL1S033Par".RecipeHeader.Cleaning.CleaningSpeed_1
      L     30; // 30%
      T     "MAL1S033Par".Par.MachineValue.SollwertFahrantrieb;
TAU2: NOP   0;
      NOP   0;
NETWORK
TITLE =ASW_9000: Step cleaning
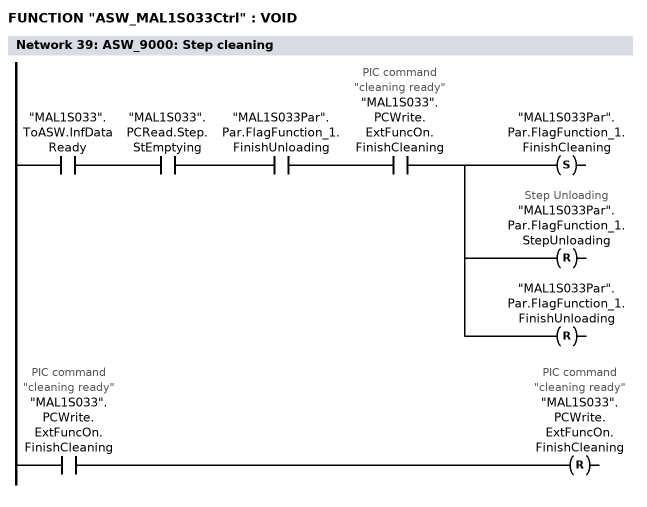

      U     "MAL1S033".ToASW.InfDataReady;
      U     "MAL1S033".PCRead.Step.StEmptying;
      U     "MAL1S033Par".Par.FlagFunction_1.FinishUnloading;
      U     "MAL1S033".PCWrite.ExtFuncOn.FinishCleaning; // PIC command "cleaning ready"
      S     "MAL1S033Par".Par.FlagFunction_1.FinishCleaning;
      R     "MAL1S033Par".Par.FlagFunction_1.StepUnloading; // Step Unloading
      R     "MAL1S033Par".Par.FlagFunction_1.FinishUnloading;
//
      U     "MAL1S033".PCWrite.ExtFuncOn.FinishCleaning; // PIC command "cleaning ready"
      R     "MAL1S033".PCWrite.ExtFuncOn.FinishCleaning; // PIC command "cleaning ready"
NETWORK
TITLE =ASW_9080: Send section date to PIC after germination

      AUF   "MAL1S033";
      U     "MAL1S033".PCRead.Step.StEmptying;
      FP    "MAL1S033Par".Par.FlagProcess.FP_SendResultToPIC;
      SPBN  E908;
//

E908: NOP   0;
NETWORK
TITLE =ASW_9099: Init Flag
////MW 2010.04.26
//-Extended section commands---
      L     0;
      T     #tmpInt;
      CALL "SIEMENS_FILL" (
           BVAL                     := #tmpInt,
           RET_VAL                  := #tmpRET,
           BLK                      := "MAL1S033".PCWrite.ExtFuncOn);

      CALL "SIEMENS_FILL" (
           BVAL                     := #tmpInt,
           RET_VAL                  := #tmpRET,
           BLK                      := "MAL1S033".PCWrite.ExtFuncOff);

NETWORK
TITLE =ASW_10000: ILO functions

      U     "MAL1S033".SecAc.Sta1On.Inf08;
      =     "MAL1S033".Gr.All.Spare04;

//- Little help for PIC-People, Number 3
      UN    "G291M".Gr.InManual; // LIFTING DEVICE KILN 2
      UN    "G292M".Gr.InManual; // TRAVELLING DRIVE KILN 2
      UN    "G293M".Gr.InManual; // UNLOADING / LOADING SCREW KILN 2
      UN    "G294M".Gr.InManual; // DISCHARGE DOOR KILN 2
      UN    "G297M".Gr.InManual; // FAN KILN 2
      UN    "G298M".Gr.InManual; // FRESH AIR LOUVER KILN 2
      UN    "G299M".Gr.InManual; // RECYCLING AIR LOUVER KILN 2
      UN    "G300M".Gr.InManual; // EXHAUST AIR LOUVER KILN 2
      UN    "G302M".Gr.InManual; // HEATING KILN 2
      UN    "G303M".Gr.InManual; // LOUVER AIR HEATER 1 FOR KILN 2
      UN    "G304M".Gr.InManual; // WITHERING AIR KILN 2
      UN    "G279M".Gr.InManual; // HEATING KILN 1 + 2
      FP    DB923.DBX 3029.0;
      =     DB923.DBX 3029.1;
      U     DB923.DBX 3029.1;
      SPBN  RSM3;
      L     0;
      T     "MAL1S033Par".Ilo.Code_ILO_Funktion0; // FCM 32 LINE 1 SEC 32 KILN
      T     "MAL1S033Par".Ilo.ILOMode;
RSM3: NOP   0;

//- Combination OLD and NEW ---
      U     "MAL1S033".SecAc.Sta1On.Inf08;
      SPBN  IFM;
      L     "MAL1S033Par".Ilo.ILOMode;
      L     100;
      *I    ;
      T     "MAL1S033Par".Ilo.Code_ILO_Funktion0;
IFM:  NOP   0;

//  no ILO-mode >> cmd manual off to all used groups and reset all flags
      U     "MAL1S033".SecAc.Sta1On.Inf08;
      FN    "MAL1S033Par".Ilo.Flag.EdgeILOModeOn;
//MW 2010.04.26      S     "MAL1S033Par".Ilo.GrCMDManOff[1]    // (ManOff)
//MW 2010.04.26      R     "MAL1S033Par".Ilo.GrCMDManAdditional.Cmd1[1]
//MW 2010.04.26      R     "MAL1S033Par".Ilo.GrCMDManAdditional.Cmd2[2]
//  Gr-cmd manual OFF
      S     "G291M".Gr.CmdManualOff; // LIFTING DEVICE KILN 2
      S     "G292M".Gr.CmdManualOff; // TRAVELLING DRIVE KILN 2
      S     "G293M".Gr.CmdManualOff; // UNLOADING / LOADING SCREW KILN 2
      S     "G294M".Gr.CmdManualOff; // DISCHARGE DOOR KILN 2
      S     "G297M".Gr.CmdManualOff; // FAN KILN 2
      S     "G298M".Gr.CmdManualOff; // FRESH AIR LOUVER KILN 2
      S     "G299M".Gr.CmdManualOff; // RECYCLING AIR FLAP KILN 2
      S     "G302M".Gr.CmdManualOff; // HEATING KILN 2
      S     "G303M".Gr.CmdManualOff; // LOUVER AIR HEATER KILN 2
      S     "G304M".Gr.CmdManualOff; // WITHERING AIR KILN 2
      S     "G305M".Gr.CmdManualOff; // CHAIN CONVEYOR 9002 KILN 2
      S     "G279M".Gr.CmdManualOff; // HEATING KILN 1 + 2
//  RESET ADDITIONAL CMD`S
      R     "G291M".USW14; // ILO-cmd
      R     "G291M".USW15; // ILO-cmd
      R     "G292M".USW14; // ILO-cmd
      R     "G292M".USW15; // ILO-cmd
      R     "G293M".USW14; // ILO-cmd
      R     "G293M".USW15; // ILO-cmd
      R     "G294M".USW14; // ILO-cmd
      R     "G294M".USW15; // ILO-cmd
      R     "G297M".USW14; // ILO-cmd
      R     "G297M".USW15; // ILO-cmd
      R     "G298M".USW14; // ILO-cmd
      R     "G298M".USW15; // ILO-cmd
      R     "G299M".USW14; // ILO-cmd
      R     "G299M".USW15; // ILO-cmd
      R     "G302M".USW14; // ILO-cmd
      R     "G302M".USW15; // ILO-cmd
      R     "G303M".USW14; // ILO-cmd
      R     "G303M".USW15; // ILO-cmd
      R     "G304M".USW14; // ILO-cmd
      R     "G304M".USW15; // ILO-cmd
      R     "G305M".USW14; // ILO-cmd
      R     "G305M".USW15; // ILO-cmd
      R     "G279M".USW14; // ILO-cmd
      R     "G279M".USW15; // ILO-cmd

//MW 2010.04.26
//- Little help for PIC-People, Number 2
      U     "MAL1S033".SecAc.Sta1On.Inf08;
      SPB   RSM2;
      L     0;
      T     #tmpInt;
      CALL "SIEMENS_FILL" (
           BVAL                     := #tmpInt,
           RET_VAL                  := #tmpRET,
           BLK                      := "MAL1S033Par".Ilo);
RSM2: NOP   0;

      NOP   0;
// --- FCM 01 - Lifting devices ---
      L     "MAL1S033Par".Ilo.ILOMode;
      L     1;
      <>I   ;
      SPB   IO1;
// man on
      U     "MAL1S033Par".Ilo.GrCMDManOn[1];
      S     "G291M".Gr.InManual; // LIFTING DEVICE KILN 2
      R     "MAL1S033Par".Ilo.GrCMDManOn[1];
// man off
      U     "MAL1S033Par".Ilo.GrCMDManOff[1];
      S     "G291M".Gr.CmdManualOff; // LIFTING DEVICE KILN 2
      R     "G291M".Gr.InManual; // LIFTING DEVICE KILN 2
      R     "G291M".USW14; // ILO-cmd
      R     "G291M".USW15; // ILO-cmd
      R     "MAL1S033Par".Ilo.GrCMDManOff[1];
      R     "MAL1S033Par".Ilo.GrCMDManAdditional.Cmd1[1];
      R     "MAL1S033Par".Ilo.GrCMDManAdditional.Cmd2[1];
// man start
      U     "MAL1S033Par".Ilo.GrCMDManStart[1];
      S     "G291M".Gr.CmdOn; // LIFTING DEVICE KILN 2
      S     "G291M".Gr.CmdContinue; // LIFTING DEVICE KILN 2
      R     "MAL1S033Par".Ilo.GrCMDManStart[1];
      U     "MAL1S033Par".Ilo.GrCMDManStart[2];
      R     "MAL1S033Par".Ilo.GrCMDManStart[2];
// man stop
      U     "MAL1S033Par".Ilo.GrCMDManStop[1];
      S     "G291M".Gr.CmdOff; // LIFTING DEVICE KILN 2
      R     "MAL1S033Par".Ilo.GrCMDManStop[1];
// man fault reset
      U     "MAL1S033Par".Ilo.GrCMDManFaultReset[1];
      S     "G291M".Gr.CmdFaultReset; // LIFTING DEVICE KILN 2
      R     "MAL1S033Par".Ilo.GrCMDManFaultReset[1];
// moving direction
      UN    "G291M".Gr.InManual; // LIFTING DEVICE KILN 2
      O(    ;
      L     "MAL1S033Par".Ilo.Code_ILO_Funktion0;
      L     100;
      <>I   ;
      )     ;
      SPB   Stat;
      UN    "MAL1S033Par".Ilo.GrCMDManAdditional.Cmd1[1];
      UN    "MAL1S033Par".Ilo.GrCMDManAdditional.Cmd2[1];
      L     "MAL1S033Par".Par.MachineValue.SOLLWERT_HUBZUG1_HOEHE;
      SPB   Tpos;
      U     "MAL1S033Par".Ilo.GrCMDManAdditional.Cmd1[1]; // ManUp
      L     2000; // 1850mm + Offset = 2000mm
      SPB   Tpos;
      U     "MAL1S033Par".Ilo.GrCMDManAdditional.Cmd2[1]; // ManDown
      L     0; // 0mm
      SPB   Tpos;
      SPA   Stat;
// target position
Tpos: NOP   0;
      T     "MAL1S033Par".Par.ParIntProcess.TarPos_ILO_LiftDev;
Stat: NOP   0;
IO1:  NOP   0;
      NOP   0;
// --- FCM 04 - Fans ---
      L     "MAL1S033Par".Ilo.ILOMode;
      L     4;
      <>I   ;
      SPB   IO4;
// man on
      U     "MAL1S033Par".Ilo.GrCMDManOn[1];
      S     "G297M".Gr.InManual; // FAN KILN 2
//MW 2010.04.26
      S     "G299M".Gr.InManual; // RECYCLING AIR LOUVER KILN 2
      S     "G299M".Gr.CmdOn; // No Button: RECYCLING AIR LOUVER KILN 2
      S     "G299M".Gr.CmdContinue; // No Button RECYCLING AIR LOUVER KILN 2
      R     "MAL1S033Par".Ilo.GrCMDManOn[1];
// man off
      U     "MAL1S033Par".Ilo.GrCMDManOff[1];
      S     "G297M".Gr.CmdManualOff; // FAN KILN 2
      R     "G297M".Gr.InManual; // FAN KILN 2
      R     "G297M".USW14; // ILO-cmd
      R     "G297M".USW15; // ILO-cmd
//MW 2010.04.26
      S     "G299M".Gr.CmdManualOff; // RECYCLING AIR LOUVER KILN 2
      R     "G299M".Gr.InManual; // RECYCLING AIR LOUVER KILN 2
      R     "G299M".USW14; // ILO-cmd
      R     "G299M".USW15; // ILO-cmd
      R     "MAL1S033Par".Ilo.GrCMDManOff[1];
      R     "MAL1S033Par".Ilo.GrCMDManAdditional.Cmd1[1];
      R     "MAL1S033Par".Ilo.GrCMDManAdditional.Cmd2[1];
// man start
      U     "MAL1S033Par".Ilo.GrCMDManStart[1];
      S     "G297M".Gr.CmdOn; // FAN KILN 2
      S     "G297M".Gr.CmdContinue; // FAN KILN 2
//MW 2010.04.26
      S     "G299M".Gr.CmdOn; // No Button: RECYCLING AIR LOUVER KILN 2
      S     "G299M".Gr.CmdContinue; // No Button RECYCLING AIR LOUVER KILN 2
      R     "MAL1S033Par".Ilo.GrCMDManStart[1];
      U     "MAL1S033Par".Ilo.GrCMDManStart[2];
      R     "MAL1S033Par".Ilo.GrCMDManStart[2];
// man stop
      U     "MAL1S033Par".Ilo.GrCMDManStop[1];
      S     "G297M".Gr.CmdOff; // FAN KILN 2
      R     "MAL1S033Par".Ilo.GrCMDManStop[1];
// man fault reset
      U     "MAL1S033Par".Ilo.GrCMDManFaultReset[1];
      S     "G297M".Gr.CmdFaultReset; // FAN KILN 2
//MW 2010.04.26
      S     "G299M".Gr.CmdFaultReset; // RECYCLING AIR LOUVER KILN 2
      R     "MAL1S033Par".Ilo.GrCMDManFaultReset[1];
// target position
      UN    "G297M".Gr.InManual; // FAN KILN 2
      O(    ;
      L     "MAL1S033Par".Ilo.Code_ILO_Funktion0;
      L     400;
      <>I   ;
      )     ;
      SPB   F04a;
      L     "MAL1S033Par".Ilo.SetpointInt01[1];
      T     "MAL1S033Par".Par.ParIntProcess.Speed_ILO_Fan;
F04a: NOP   0;
//MW 2010.04.26
      UN    "G299M".Gr.InManual; // Recycling Air Flap Kilningbox 2
      O(    ;
      L     "MAL1S033Par".Ilo.Code_ILO_Funktion0;
      L     400;
      <>I   ;
      )     ;
      SPB   F04b;
//MW      L     90                          // 90%
      L     100; // 100%
      T     "MAL1S033Par".Par.ParIntProcess.TarPos_ILO_RecycAir;
F04b: NOP   0;

IO4:  NOP   0;
      NOP   0;
// --- FCM 05 - Fans with target air temperature ---
      L     "MAL1S033Par".Ilo.ILOMode;
      L     5;
      <>I   ;
      SPB   IO5;
// man on
      U     "MAL1S033Par".Ilo.GrCMDManOn[1];
      S     "G297M".Gr.InManual; // FAN KILN 2
      S     "G299M".Gr.InManual; // RECYCLING AIR FLAP KILN 2
      S     "G299M".Gr.CmdOn; // No Button: RECYCLING AIR FLAP KILN 2
      S     "G299M".Gr.CmdContinue; // No Button RECYCLING AIR FLAP KILN 2
      S     "G302M".Gr.InManual; // HEATING KILN 2
      S     "G302M".Gr.CmdOn; // No Button: HEATING KILN 2
      S     "G302M".Gr.CmdContinue; // No Button HEATING KILN 2
      S     "G303M".Gr.InManual; // LOUVER AIR HEATER KILN 2
      S     "G303M".Gr.CmdOn; // No Button: LOUVER AIR HEATER KILN 2
      S     "G303M".Gr.CmdContinue; // No Button LOUVER AIR HEATER KILN 2
//MW 2010.04.26      S     "G298M".Gr.InManual         // FRESH AIR LOUVER KILN 2
//MW 2010.04.26      S     "G298M".Gr.CmdOn            // No Button: FRESH AIR LOUVER KILN 2
//MW 2010.04.26      S     "G298M".Gr.CmdContinue      // No Button FRESH AIR LOUVER KILN 2
      S     "G304M".Gr.InManual; // WITHERING AIR KILN 2
      S     "G304M".Gr.CmdOn; // No Button: WITHERING AIR KILN 2
      S     "G304M".Gr.CmdContinue; // No Button WITHERING AIR KILN 2
      R     "MAL1S033Par".Ilo.GrCMDManOn[1];
// man off
      U     "MAL1S033Par".Ilo.GrCMDManOff[1];
      S     "G297M".Gr.CmdManualOff; // FAN KILN 2
      R     "G297M".Gr.InManual; // FAN KILN 2
      R     "G297M".USW14; // ILO-cmd
      R     "G297M".USW15; // ILO-cmd
      S     "G299M".Gr.CmdManualOff; // RECYCLING AIR FLAP KILN 2
      R     "G299M".Gr.InManual; // RECYCLING AIR FLAP KILN 2
      R     "G299M".USW14; // ILO-cmd
      R     "G299M".USW15; // ILO-cmd
      S     "G302M".Gr.CmdManualOff; // HEATING KILN 2
      R     "G302M".Gr.InManual; // HEATING KILN 2
      R     "G302M".USW14; // ILO-cmd
      R     "G302M".USW15; // ILO-cmd
      S     "G303M".Gr.CmdManualOff; // LOUVER AIR HEATER KILN 2
      R     "G303M".Gr.InManual; // LOUVER AIR HEATER KILN 2
      R     "G303M".USW14; // ILO-cmd
      R     "G303M".USW15; // ILO-cmd
//MW 2010.04.26      S     "G298M".Gr.CmdManualOff     // FRESH AIR LOUVER KILN 2
//MW 2010.04.26      R     "G298M".Gr.InManual         // FRESH AIR LOUVER KILN 2
      R     "G298M".USW14; // ILO-cmd
      R     "G298M".USW15; // ILO-cmd
      S     "G304M".Gr.CmdManualOff; // WITHERING AIR KILN 2
      R     "G304M".Gr.InManual; // WITHERING AIR KILN 2
      R     "G304M".USW14; // ILO-cmd
      R     "G304M".USW15; // ILO-cmd
      R     "MAL1S033Par".Ilo.GrCMDManOff[1];
      R     "MAL1S033Par".Ilo.GrCMDManAdditional.Cmd1[1];
      R     "MAL1S033Par".Ilo.GrCMDManAdditional.Cmd2[1];
// man start
      U     "MAL1S033Par".Ilo.GrCMDManStart[1];
      S     "G297M".Gr.CmdOn; // FAN KILN 2
      S     "G297M".Gr.CmdContinue; // FAN KILN 2
      S     "G299M".Gr.CmdOn; // RECYCLING AIR FLAP KILN 2
      S     "G299M".Gr.CmdContinue; // RECYCLING AIR FLAP KILN 2
      S     "G302M".Gr.CmdOn; // HEATING KILN 2
      S     "G302M".Gr.CmdContinue; // HEATING KILN 2
      S     "G303M".Gr.CmdOn; // LOUVER AIR HEATER KILN 2
      S     "G303M".Gr.CmdContinue; // LOUVER AIR HEATER KILN 2
//MW 2010.04.26      S     "G298M".Gr.CmdOn            // FRESH AIR LOUVER KILN 2
//MW 2010.04.26      S     "G298M".Gr.CmdContinue      // FRESH AIR LOUVER KILN 2
      S     "G304M".Gr.CmdOn; // WITHERING AIR KILN 2
      S     "G304M".Gr.CmdContinue; // WITHERING AIR KILN 2
      R     "MAL1S033Par".Ilo.GrCMDManStart[1];
      U     "MAL1S033Par".Ilo.GrCMDManStart[2];
      R     "MAL1S033Par".Ilo.GrCMDManStart[2];
// man stop
//MW 2010.04.26      U     "MAL1S033Par".Ilo.GrSTMan[17]
      U     "MAL1S033Par".Ilo.GrCMDManStop[1];
      S     "G297M".Gr.CmdOff; // FAN KILN 2
      S     "G299M".Gr.CmdOff; // RECYCLING AIR FLAP KILN 2
      S     "G302M".Gr.CmdOff; // HEATING KILN 2
      S     "G303M".Gr.CmdOff; // LOUVER AIR HEATER KILN 2
//MW 2010.04.26      S     "G298M".Gr.CmdOff           // FRESH AIR LOUVER KILN 2
      S     "G304M".Gr.CmdOff; // WITHERING AIR KILN 2
//MW 2010.04.26      R     "MAL1S033Par".Ilo.GrSTMan[17]
      R     "MAL1S033Par".Ilo.GrCMDManStop[1];
// man fault reset
      U     "MAL1S033Par".Ilo.GrCMDManFaultReset[1];
      S     "G297M".Gr.CmdFaultReset; // FAN KILN 2
      S     "G299M".Gr.CmdFaultReset; // RECYCLING AIR FLAP KILN 2
      S     "G302M".Gr.CmdFaultReset; // HEATING KILN 2
      S     "G303M".Gr.CmdFaultReset; // LOUVER AIR HEATER KILN 2
//MW 2010.04.26      S     "G298M".Gr.CmdFaultReset    // FRESH AIR LOUVER KILN 2
      S     "G304M".Gr.CmdFaultReset; // WITHERING AIR KILN 2
      R     "MAL1S033Par".Ilo.GrCMDManFaultReset[1];
// target position
      UN    "G297M".Gr.InManual; // FAN KILN 2
      O(    ;
      L     "MAL1S033Par".Ilo.Code_ILO_Funktion0;
      L     500;
      <>I   ;
      )     ;
      SPB   F05b;
      L     "MAL1S033Par".Ilo.SetpointInt01[1];
      T     "MAL1S033Par".Par.ParIntProcess.Speed_ILO_Fan;
F05b: NOP   0;
      UN    "G299M".Gr.InManual; // Recycling Air Flap Kilningbox 1
      O(    ;
      L     "MAL1S033Par".Ilo.Code_ILO_Funktion0;
      L     500;
      <>I   ;
      )     ;
      SPB   F05c;
      L     "MAL1S033Par".Ilo.SetpointInt03[1];
      T     "MAL1S033Par".Par.ParIntProcess.TarPos_ILO_RecycAir;
F05c: NOP   0;
      UN    "G304M".Gr.InManual; // Withering Air Flap Kilningbox 1
      O(    ;
      L     "MAL1S033Par".Ilo.Code_ILO_Funktion0;
      L     500;
      <>I   ;
      )     ;
      SPB   F05d;
      L     "MAL1S033Par".Ilo.SetpointInt04[1];
      T     "MAL1S033Par".Par.ParIntProcess.TarPos_ILO_WitheringAir;
F05d: NOP   0;
      UN    "G302M".Gr.InManual; // Heating Kiln 2
      O(    ;
      L     "MAL1S033Par".Ilo.Code_ILO_Funktion0;
      L     500;
      <>I   ;
      )     ;
      SPB   F05e;
//MW 2010.04.26      L     "MAL1S033Par".Ilo.SetpointInt01[2]
      L     "MAL1S033Par".Ilo.SetpointInt02[1];
      T     "MAL1S033Par".Par.ParIntProcess.TargetTemperature_ILO;
F05e: NOP   0;

IO5:  NOP   0;
      NOP   0;
// --- FCM 06 - Fresh air flap ---
      L     "MAL1S033Par".Ilo.ILOMode;
      L     6;
      <>I   ;
      SPB   IO6;
// man on
      U     "MAL1S033Par".Ilo.GrCMDManOn[1];
      S     "G298M".Gr.InManual; // FRESH AIR LOUVER KILN 2
      R     "MAL1S033Par".Ilo.GrCMDManOn[1];
// man off
      U     "MAL1S033Par".Ilo.GrCMDManOff[1];
      S     "G298M".Gr.CmdManualOff; // FRESH AIR LOUVER KILN 2
      R     "G298M".Gr.InManual; // FRESH AIR LOUVER KILN 2
      R     "G298M".USW14; // ILO-cmd
      R     "G298M".USW15; // ILO-cmd
      R     "MAL1S033Par".Ilo.GrCMDManOff[1];
      R     "MAL1S033Par".Ilo.GrCMDManAdditional.Cmd1[1];
      R     "MAL1S033Par".Ilo.GrCMDManAdditional.Cmd2[1];
// man start
      U     "MAL1S033Par".Ilo.GrCMDManStart[1];
      S     "G298M".Gr.CmdOn; // FRESH AIR LOUVER KILN 2
      S     "G298M".Gr.CmdContinue; // FRESH AIR LOUVER KILN 2
      R     "MAL1S033Par".Ilo.GrCMDManStart[1];
      U     "MAL1S033Par".Ilo.GrCMDManStart[2];
      R     "MAL1S033Par".Ilo.GrCMDManStart[2];
// man stop
      U     "MAL1S033Par".Ilo.GrCMDManStop[1];
      S     "G298M".Gr.CmdOff; // FRESH AIR LOUVER KILN 2
      R     "MAL1S033Par".Ilo.GrCMDManStop[1];
// man fault reset
      U     "MAL1S033Par".Ilo.GrCMDManFaultReset[1];
      S     "G298M".Gr.CmdFaultReset; // FRESH AIR LOUVER KILN 2
      R     "MAL1S033Par".Ilo.GrCMDManFaultReset[1];
// moving direction

// target position
      UN    "G298M".Gr.InManual; // FRESH AIR LOUVER KILN 2
      SPB   F06b;
      L     "MAL1S033Par".Ilo.SetpointInt01[1];
      T     "MAL1S033Par".Par.ParIntProcess.TarPos_ILO_FreshAir;
F06b: NOP   0;

IO6:  NOP   0;
      NOP   0;
// --- FCM 07 - Recycling air flap ---
      L     "MAL1S033Par".Ilo.ILOMode;
      L     7;
      <>I   ;
      SPB   IO7;
// man on
      U     "MAL1S033Par".Ilo.GrCMDManOn[1];
      S     "G299M".Gr.InManual; // RECYCLING AIR FLAP KILN 2
      S     "G304M".Gr.InManual; // WITHERING AIR KILN 2
      R     "MAL1S033Par".Ilo.GrCMDManOn[1];
// man off
      U     "MAL1S033Par".Ilo.GrCMDManOff[1];
      S     "G299M".Gr.CmdManualOff; // RECYCLING AIR FLAP KILN 2
      R     "G299M".Gr.InManual; // RECYCLING AIR FLAP KILN 2
      R     "G299M".USW14; // ILO-cmd
      R     "G299M".USW15; // ILO-cmd
      S     "G304M".Gr.CmdManualOff; // WITHERING AIR KILN 2
      R     "G304M".Gr.InManual; // WITHERING AIR KILN 2
      R     "G304M".USW14; // ILO-cmd
      R     "G304M".USW15; // ILO-cmd
      R     "MAL1S033Par".Ilo.GrCMDManOff[1];
      R     "MAL1S033Par".Ilo.GrCMDManAdditional.Cmd1[1];
      R     "MAL1S033Par".Ilo.GrCMDManAdditional.Cmd2[1];
// man start
      U     "MAL1S033Par".Ilo.GrCMDManStart[1];
      S     "G299M".Gr.CmdOn; // RECYCLING AIR FLAP KILN 2
      S     "G299M".Gr.CmdContinue; // RECYCLING AIR FLAP KILN 2
      S     "G304M".Gr.CmdOn; // WITHERING AIR KILN 2
      S     "G304M".Gr.CmdContinue; // WITHERING AIR KILN 2
      R     "MAL1S033Par".Ilo.GrCMDManStart[1];
      U     "MAL1S033Par".Ilo.GrCMDManStart[2];
      R     "MAL1S033Par".Ilo.GrCMDManStart[2];
// man stop
      U     "MAL1S033Par".Ilo.GrCMDManStop[1];
      S     "G299M".Gr.CmdOff; // RECYCLING AIR FLAP KILN 2
      S     "G304M".Gr.CmdOff; // WITHERING AIR KILN 2
      R     "MAL1S033Par".Ilo.GrCMDManStop[1];
// man fault reset
      U     "MAL1S033Par".Ilo.GrCMDManFaultReset[1];
      S     "G299M".Gr.CmdFaultReset; // RECYCLING AIR FLAP KILN 2
      S     "G304M".Gr.CmdFaultReset; // WITHERING AIR KILN 2
      R     "MAL1S033Par".Ilo.GrCMDManFaultReset[1];
// moving direction

// target position
      UN    "G299M".Gr.InManual; // RECYCLING AIR FLAP KILN 2
      SPB   F07a;
      L     "MAL1S033Par".Ilo.SetpointInt01[1];
      T     "MAL1S033Par".Par.ParIntProcess.TarPos_ILO_RecycAir;
F07a: NOP   0;
IO7:  NOP   0;
      NOP   0;
// --- FCM 09 - Floor drives ---
      L     "MAL1S033Par".Ilo.ILOMode;
      L     9;
      <>I   ;
      SPB   IO9;
// man on
      U     "MAL1S033Par".Ilo.GrCMDManOn[1];
      S     "G292M".Gr.InManual; // TRAVELLING DRIVE KILN 2
      R     "MAL1S033Par".Ilo.GrCMDManOn[1];
// man off
      U     "MAL1S033Par".Ilo.GrCMDManOff[1];
      S     "G292M".Gr.CmdManualOff; // TRAVELLING DRIVE KILN 2
      R     "G292M".Gr.InManual; // TRAVELLING DRIVE KILN 2
      R     "G292M".USW14; // ILO-cmd
      R     "G292M".USW15; // ILO-cmd
      R     "MAL1S033Par".Ilo.GrCMDManOff[1];
      R     "MAL1S033Par".Ilo.GrCMDManAdditional.Cmd1[1];
      R     "MAL1S033Par".Ilo.GrCMDManAdditional.Cmd2[1];
// man start
      U     "MAL1S033Par".Ilo.GrCMDManStart[1];
      S     "G292M".Gr.CmdOn; // TRAVELLING DRIVE KILN 2
      S     "G292M".Gr.CmdContinue; // TRAVELLING DRIVE KILN 2
      R     "MAL1S033Par".Ilo.GrCMDManStart[1];
      U     "MAL1S033Par".Ilo.GrCMDManStart[2];
      R     "MAL1S033Par".Ilo.GrCMDManStart[2];
// man stop
      U     "MAL1S033Par".Ilo.GrCMDManStop[1];
      S     "G292M".Gr.CmdOff; // TRAVELLING DRIVE KILN 2
      R     "MAL1S033Par".Ilo.GrCMDManStop[1];
// man fault reset
      U     "MAL1S033Par".Ilo.GrCMDManFaultReset[1];
      S     "G292M".Gr.CmdFaultReset; // TRAVELLING DRIVE KILN 2
      R     "MAL1S033Par".Ilo.GrCMDManFaultReset[1];
      NOP   0;
      UN    "G292M".Gr.InManual; // TRAVELLING DRIVE KILN 2
      O     ;
      UN    "MAL1S033Par".Ilo.GrCMDManAdditional.Cmd1[1];
      UN    "MAL1S033Par".Ilo.GrCMDManAdditional.Cmd2[1];
      SPB   f092;
      U     "MAL1S033Par".Ilo.GrCMDManAdditional.Cmd1[1];
      =     "G292M".USW14; // ILO-cmd run fwd
      U     "MAL1S033Par".Ilo.GrCMDManAdditional.Cmd2[1];
      =     "G292M".USW15; // ILO-cmd run rev
// target position
      L     "MAL1S033Par".Ilo.SetpointInt01[1];
      T     "MAL1S033Par".Par.ParIntProcess.Speed_ILO_FloorRotating;
f092: NOP   0;

IO9:  NOP   0;
      NOP   0;
// --- FCM 10 - Floor drives and lifting devices ---
      L     "MAL1S033Par".Ilo.ILOMode;
      L     10;
      <>I   ;
      SPB   IO10;
// man on
      U     "MAL1S033Par".Ilo.GrCMDManOn[1];
      S     "G291M".Gr.InManual; // LIFTING DEVICE KILN 2
      S     "G291M".Gr.CmdOn; // No Button: LIFTING DEVICE KILN 2
      S     "G291M".Gr.CmdContinue; // No Button LIFTING DEVICE KILN 2
      S     "G292M".Gr.InManual; // TRAVELLING DRIVE KILN 2
      R     "MAL1S033Par".Ilo.GrCMDManOn[1];
// man off
      U     "MAL1S033Par".Ilo.GrCMDManOff[1];
      S     "G291M".Gr.CmdManualOff; // LIFTING DEVICE KILN 2
      R     "G291M".Gr.InManual; // LIFTING DEVICE KILN 2
      R     "G291M".USW14; // ILO-cmd
      R     "G291M".USW15; // ILO-cmd
      S     "G292M".Gr.CmdManualOff; // TRAVELLING DRIVE KILN 2
      R     "G292M".Gr.InManual; // TRAVELLING DRIVE KILN 2
      R     "G292M".USW14; // ILO-cmd
      R     "G292M".USW15; // ILO-cmd
      R     "MAL1S033Par".Ilo.GrCMDManOff[1];
      R     "MAL1S033Par".Ilo.GrCMDManAdditional.Cmd1[1];
      R     "MAL1S033Par".Ilo.GrCMDManAdditional.Cmd2[1];
// man start
      U     "MAL1S033Par".Ilo.GrCMDManStart[1];
      S     "G292M".Gr.CmdOn; // TRAVELLING DRIVE KILN 2
      S     "G292M".Gr.CmdContinue; // TRAVELLING DRIVE KILN 2
      R     "MAL1S033Par".Ilo.GrCMDManStart[1];
      U     "MAL1S033Par".Ilo.GrCMDManStart[2];
      S     "G291M".Gr.CmdOn; // LIFTING DEVICE KILN 2
      S     "G291M".Gr.CmdContinue; // LIFTING DEVICE KILN 2
      R     "MAL1S033Par".Ilo.GrCMDManStart[2];
      U     "MAL1S033Par".Ilo.GrCMDManStart[3];
      R     "MAL1S033Par".Ilo.GrCMDManStart[3];
// man stop
      U     "MAL1S033Par".Ilo.GrCMDManStop[1];
      S     "G291M".Gr.CmdOff; // LIFTING DEVICE KILN 2
      S     "G292M".Gr.CmdOff; // TRAVELLING DRIVE KILN 2
      R     "MAL1S033Par".Ilo.GrCMDManStop[1];
// man fault reset
      U     "MAL1S033Par".Ilo.GrCMDManFaultReset[1];
      S     "G291M".Gr.CmdFaultReset; // LIFTING DEVICE KILN 2
      S     "G292M".Gr.CmdFaultReset; // TRAVELLING DRIVE KILN 2
      R     "MAL1S033Par".Ilo.GrCMDManFaultReset[1];
// moving direction
      NOP   0;
      UN    "G292M".Gr.InManual; // TRAVELLING DRIVE KILN 2
      O     ;
      UN    "MAL1S033Par".Ilo.GrCMDManAdditional.Cmd1[1];
      UN    "MAL1S033Par".Ilo.GrCMDManAdditional.Cmd2[1];
      SPB   f102;
      U     "MAL1S033Par".Ilo.GrCMDManAdditional.Cmd1[1];
      =     "G292M".USW14; // ILO-cmd run fwd
      U     "MAL1S033Par".Ilo.GrCMDManAdditional.Cmd2[1];
      =     "G292M".USW15; // ILO-cmd run rev
// target speed floor drives
      L     "MAL1S033Par".Ilo.SetpointInt01[1];
      T     "MAL1S033Par".Par.ParIntProcess.Speed_ILO_FloorRotating;
f102: NOP   0;
      UN    "G291M".Gr.InManual; // LIFTING DEVICE KILN 2
      O(    ;
      L     "MAL1S033Par".Ilo.Code_ILO_Funktion0;
      L     1000;
      <>I   ;
      )     ;
      SPB   f103;
// target position lifting devices
      L     "MAL1S033Par".Ilo.SetpointInt02[1];
      T     "MAL1S033Par".Par.ParIntProcess.TarPos_ILO_LiftDev;
f103: NOP   0;

